    movel([0.122327, -1.228329, -2.662622, -0.821438, 1.570796, 1.693123],accel_mss,speed_ms,0,blend_radius_m)
    movel([0.122064, -1.229821, -2.661862, -0.820705, 1.570796, 1.692861],accel_mss,speed_ms,0,blend_radius_m)
    movel([0.121775, -1.231117, -2.661201, -0.820072, 1.570796, 1.692571],accel_mss,speed_ms,0,blend_radius_m)
    movel([0.121353, -1.232704, -2.660387, -0.819297, 1.570796, 1.692149],accel_mss,speed_ms,0,blend_radius_m)
    movel([0.120445, -1.235790, -2.658798, -0.817801, 1.570796, 1.691242],accel_mss,speed_ms,0,blend_radius_m)
    speed_ms = 0.003
    movel([0.120445, -1.239413, -2.660528, -0.812448, 1.570796, 1.691242],accel_mss,speed_ms,0,blend_radius_m)
    speed_ms = 0.007
    movel([0.119507, -1.242259, -2.659045, -0.811085, 1.570796, 1.690304],accel_mss,speed_ms,0,blend_radius_m)
    movel([0.118536, -1.244874, -2.657674, -0.809842, 1.570796, 1.689333],accel_mss,speed_ms,0,blend_radius_m)
    movel([0.117534, -1.247261, -2.656415, -0.808713, 1.570796, 1.688331],accel_mss,speed_ms,0,blend_radius_m)
    movel([0.117009, -1.248417, -2.655802, -0.808169, 1.570796, 1.687805],accel_mss,speed_ms,0,blend_radius_m)
    movel([0.116695, -1.249022, -2.655481, -0.807885, 1.570796, 1.687491],accel_mss,speed_ms,0,blend_radius_m)
    movel([0.116436, -1.249403, -2.655279, -0.807707, 1.570796, 1.687232],accel_mss,speed_ms,0,blend_radius_m)
    movel([0.116154, -1.249681, -2.655131, -0.807576, 1.570796, 1.686950],accel_mss,speed_ms,0,blend_radius_m)
    movel([0.114416, -1.250711, -2.654583, -0.807095, 1.570796, 1.685212],accel_mss,speed_ms,0,blend_radius_m)
    movel([0.110469, -1.252305, -2.653732, -0.806351, 1.570796, 1.681265],accel_mss,speed_ms,0,blend_radius_m)
    movel([0.105892, -1.253965, -2.652843, -0.805581, 1.570796, 1.676688],accel_mss,speed_ms,0,blend_radius_m)
    movel([0.101275, -1.255432, -2.652054, -0.804903, 1.570796, 1.672071],accel_mss,speed_ms,0,blend_radius_m)
    movel([0.097010, -1.256607, -2.651420, -0.804361, 1.570796, 1.667806],accel_mss,speed_ms,0,blend_radius_m)
    movel([0.093314, -1.257431, -2.650975, -0.803983, 1.570796, 1.664111],accel_mss,speed_ms,0,blend_radius_m)
    movel([0.090388, -1.257913, -2.650714, -0.803762, 1.570796, 1.661185],accel_mss,speed_ms,0,blend_radius_m)
    movel([0.089540, -1.257658, -2.650852, -0.803879, 1.570796, 1.660336],accel_mss,speed_ms,0,blend_radius_m)
    movel([0.088883, -1.255617, -2.651955, -0.804818, 1.570796, 1.659679],accel_mss,speed_ms,0,blend_radius_m)
    movel([0.089050, -1.247881, -2.656087, -0.808421, 1.570796, 1.659846],accel_mss,speed_ms,0,blend_radius_m)
    movel([0.089536, -1.239986, -2.660230, -0.812173, 1.570796, 1.660332],accel_mss,speed_ms,0,blend_radius_m)
    movel([0.090414, -1.234541, -2.663045, -0.814803, 1.570796, 1.661211],accel_mss,speed_ms,0,blend_radius_m)
    movel([0.090708, -1.233537, -2.663560, -0.815292, 1.570796, 1.661505],accel_mss,speed_ms,0,blend_radius_m)
    movel([0.091054, -1.232965, -2.663853, -0.815571, 1.570796, 1.661850],accel_mss,speed_ms,0,blend_radius_m)
    movel([0.091650, -1.232455, -2.664114, -0.815820, 1.570796, 1.662446],accel_mss,speed_ms,0,blend_radius_m)
    movel([0.093003, -1.231626, -2.664538, -0.816226, 1.570796, 1.663799],accel_mss,speed_ms,0,blend_radius_m)
    movel([0.095187, -1.230416, -2.665154, -0.816819, 1.570796, 1.665983],accel_mss,speed_ms,0,blend_radius_m)
    movel([0.097230, -1.229430, -2.665656, -0.817304, 1.570796, 1.668026],accel_mss,speed_ms,0,blend_radius_m)
    movel([0.099701, -1.228404, -2.666176, -0.817809, 1.570796, 1.670497],accel_mss,speed_ms,0,blend_radius_m)
    movel([0.103416, -1.227010, -2.666881, -0.818498, 1.570796, 1.674212],accel_mss,speed_ms,0,blend_radius_m)
    movel([0.108750, -1.225175, -2.667806, -0.819408, 1.570796, 1.679546],accel_mss,speed_ms,0,blend_radius_m)
    movel([0.113497, -1.223771, -2.668511, -0.820108, 1.570796, 1.684294],accel_mss,speed_ms,0,blend_radius_m)
    movel([0.117730, -1.222780, -2.669007, -0.820602, 1.570796, 1.688526],accel_mss,speed_ms,0,blend_radius_m)
    movel([0.121518, -1.222181, -2.669306, -0.820902, 1.570796, 1.692314],accel_mss,speed_ms,0,blend_radius_m)
    movel([0.122546, -1.222114, -2.669340, -0.820935, 1.570796, 1.693342],accel_mss,speed_ms,0,blend_radius_m)
    movel([0.122998, -1.222262, -2.669266, -0.820861, 1.570796, 1.693794],accel_mss,speed_ms,0,blend_radius_m)
    movel([0.123197, -1.222684, -2.669055, -0.820650, 1.570796, 1.693993],accel_mss,speed_ms,0,blend_radius_m)
    movel([0.123242, -1.223715, -2.668539, -0.820135, 1.570796, 1.694038],accel_mss,speed_ms,0,blend_radius_m)
    movel([0.123245, -1.224244, -2.668274, -0.819872, 1.570796, 1.694042],accel_mss,speed_ms,0,blend_radius_m)
    movel([0.123250, -1.224722, -2.668033, -0.819633, 1.570796, 1.694046],accel_mss,speed_ms,0,blend_radius_m)
    movel([0.123256, -1.225120, -2.667833, -0.819435, 1.570796, 1.694052],accel_mss,speed_ms,0,blend_radius_m)
    movel([0.123267, -1.225404, -2.667691, -0.819294, 1.570796, 1.694063],accel_mss,speed_ms,0,blend_radius_m)
    movel([0.123104, -1.226608, -2.667084, -0.818697, 1.570796, 1.693901],accel_mss,speed_ms,0,blend_radius_m)
    movel([0.122915, -1.227989, -2.666386, -0.818014, 1.570796, 1.693712],accel_mss,speed_ms,0,blend_radius_m)
    movel([0.122686, -1.229588, -2.665575, -0.817226, 1.570796, 1.693482],accel_mss,speed_ms,0,blend_radius_m)
    movel([0.122327, -1.231965, -2.664364, -0.816060, 1.570796, 1.693123],accel_mss,speed_ms,0,blend_radius_m)
    movel([0.122064, -1.233455, -2.663602, -0.815332, 1.570796, 1.692861],accel_mss,speed_ms,0,blend_radius_m)
    movel([0.121775, -1.234748, -2.662939, -0.814703, 1.570796, 1.692571],accel_mss,speed_ms,0,blend_radius_m)
    movel([0.121353, -1.236333, -2.662123, -0.813934, 1.570796, 1.692149],accel_mss,speed_ms,0,blend_radius_m)
    movel([0.120445, -1.239413, -2.660528, -0.812448, 1.570796, 1.691242],accel_mss,speed_ms,0,blend_radius_m)
    speed_ms = 0.003
    movel([0.120445, -1.225115, -2.653559, -0.833714, 1.570796, 1.691242],accel_mss,speed_ms,0,blend_radius_m)
    speed_ms = 1.000
    movel([0.120445, -1.198045, -2.639248, -0.875095, 1.570796, 1.691242],accel_mss,speed_ms,0,blend_radius_m)
    movel([0.119134, -1.211134, -2.632724, -0.868530, 1.570796, 1.689930],accel_mss,speed_ms,0,blend_radius_m)
    movel([0.119134, -1.238074, -2.646863, -0.827452, 1.570796, 1.689930],accel_mss,speed_ms,0,blend_radius_m)
    speed_ms = 0.003
    movel([0.119134, -1.248685, -2.652035, -0.811669, 1.570796, 1.689930],accel_mss,speed_ms,0,blend_radius_m)
    speed_ms = 0.007
    movel([0.119613, -1.248514, -2.652126, -0.811749, 1.570796, 1.690410],accel_mss,speed_ms,0,blend_radius_m)
    movel([0.120288, -1.248305, -2.652237, -0.811847, 1.570796, 1.691084],accel_mss,speed_ms,0,blend_radius_m)
    movel([0.121252, -1.248036, -2.652380, -0.811973, 1.570796, 1.692048],accel_mss,speed_ms,0,blend_radius_m)
    movel([0.122082, -1.247811, -2.652500, -0.812078, 1.570796, 1.692879],accel_mss,speed_ms,0,blend_radius_m)
    movel([0.122838, -1.247602, -2.652610, -0.812176, 1.570796, 1.693634],accel_mss,speed_ms,0,blend_radius_m)
    movel([0.123475, -1.247426, -2.652704, -0.812259, 1.570796, 1.694272],accel_mss,speed_ms,0,blend_radius_m)
    movel([0.124143, -1.247295, -2.652773, -0.812320, 1.570796, 1.694939],accel_mss,speed_ms,0,blend_radius_m)
    movel([0.124365, -1.247460, -2.652686, -0.812243, 1.570796, 1.695162],accel_mss,speed_ms,0,blend_radius_m)
    movel([0.124402, -1.247921, -2.652442, -0.812027, 1.570796, 1.695199],accel_mss,speed_ms,0,blend_radius_m)
    movel([0.124242, -1.248885, -2.651929, -0.811575, 1.570796, 1.695039],accel_mss,speed_ms,0,blend_radius_m)
    movel([0.124101, -1.249513, -2.651594, -0.811282, 1.570796, 1.694897],accel_mss,speed_ms,0,blend_radius_m)
    movel([0.123892, -1.250271, -2.651190, -0.810928, 1.570796, 1.694688],accel_mss,speed_ms,0,blend_radius_m)
    movel([0.123656, -1.251037, -2.650780, -0.810572, 1.570796, 1.694453],accel_mss,speed_ms,0,blend_radius_m)
    movel([0.123426, -1.251690, -2.650431, -0.810268, 1.570796, 1.694222],accel_mss,speed_ms,0,blend_radius_m)
    movel([0.122892, -1.252969, -2.649744, -0.809675, 1.570796, 1.693688],accel_mss,speed_ms,0,blend_radius_m)
    movel([0.122475, -1.253530, -2.649443, -0.809416, 1.570796, 1.693271],accel_mss,speed_ms,0,blend_radius_m)
    movel([0.121856, -1.253929, -2.649229, -0.809232, 1.570796, 1.692652],accel_mss,speed_ms,0,blend_radius_m)
    movel([0.120346, -1.254514, -2.648913, -0.808962, 1.570796, 1.691142],accel_mss,speed_ms,0,blend_radius_m)
    movel([0.119442, -1.254834, -2.648741, -0.808814, 1.570796, 1.690239],accel_mss,speed_ms,0,blend_radius_m)
    movel([0.118839, -1.255024, -2.648638, -0.808727, 1.570796, 1.689635],accel_mss,speed_ms,0,blend_radius_m)
    movel([0.118432, -1.255127, -2.648583, -0.808679, 1.570796, 1.689228],accel_mss,speed_ms,0,blend_radius_m)
    movel([0.118168, -1.254986, -2.648659, -0.808744, 1.570796, 1.688964],accel_mss,speed_ms,0,blend_radius_m)
    movel([0.118162, -1.254671, -2.648828, -0.808889, 1.570796, 1.688958],accel_mss,speed_ms,0,blend_radius_m)
    movel([0.118223, -1.254120, -2.649125, -0.809143, 1.570796, 1.689019],accel_mss,speed_ms,0,blend_radius_m)
    movel([0.118394, -1.253069, -2.649691, -0.809629, 1.570796, 1.689190],accel_mss,speed_ms,0,blend_radius_m)
    movel([0.118522, -1.252242, -2.650135, -0.810012, 1.570796, 1.689318],accel_mss,speed_ms,0,blend_radius_m)
    movel([0.118632, -1.251377, -2.650599, -0.810414, 1.570796, 1.689429],accel_mss,speed_ms,0,blend_radius_m)
    movel([0.118710, -1.250595, -2.651017, -0.810777, 1.570796, 1.689506],accel_mss,speed_ms,0,blend_radius_m)
    movel([0.118739, -1.250054, -2.651306, -0.811030, 1.570796, 1.689536],accel_mss,speed_ms,0,blend_radius_m)
    movel([0.118758, -1.249526, -2.651587, -0.811276, 1.570796, 1.689555],accel_mss,speed_ms,0,blend_radius_m)
    movel([0.118795, -1.249184, -2.651769, -0.811435, 1.570796, 1.689591],accel_mss,speed_ms,0,blend_radius_m)
    movel([0.118957, -1.248800, -2.651974, -0.811615, 1.570796, 1.689753],accel_mss,speed_ms,0,blend_radius_m)
    speed_ms = 0.003
    movel([0.119134, -1.252285, -2.653743, -0.806361, 1.570796, 1.689930],accel_mss,speed_ms,0,blend_radius_m)
    speed_ms = 0.007
    movel([0.119613, -1.252114, -2.653835, -0.806441, 1.570796, 1.690410],accel_mss,speed_ms,0,blend_radius_m)
    movel([0.120288, -1.251906, -2.653946, -0.806538, 1.570796, 1.691084],accel_mss,speed_ms,0,blend_radius_m)
    movel([0.121252, -1.251637, -2.654090, -0.806663, 1.570796, 1.692048],accel_mss,speed_ms,0,blend_radius_m)
    movel([0.122082, -1.251413, -2.654209, -0.806767, 1.570796, 1.692879],accel_mss,speed_ms,0,blend_radius_m)
    movel([0.122838, -1.251204, -2.654320, -0.806864, 1.570796, 1.693634],accel_mss,speed_ms,0,blend_radius_m)
    movel([0.123475, -1.251028, -2.654414, -0.806947, 1.570796, 1.694272],accel_mss,speed_ms,0,blend_radius_m)
    movel([0.124143, -1.250898, -2.654484, -0.807008, 1.570796, 1.694939],accel_mss,speed_ms,0,blend_radius_m)
    movel([0.124365, -1.251062, -2.654396, -0.806931, 1.570796, 1.695162],accel_mss,speed_ms,0,blend_radius_m)
    movel([0.124402, -1.251522, -2.654151, -0.806716, 1.570796, 1.695199],accel_mss,speed_ms,0,blend_radius_m)
    movel([0.124242, -1.252485, -2.653636, -0.806268, 1.570796, 1.695039],accel_mss,speed_ms,0,blend_radius_m)
    movel([0.124101, -1.253111, -2.653301, -0.805977, 1.570796, 1.694897],accel_mss,speed_ms,0,blend_radius_m)
    movel([0.123892, -1.253868, -2.652895, -0.805626, 1.570796, 1.694688],accel_mss,speed_ms,0,blend_radius_m)
    movel([0.123656, -1.254633, -2.652484, -0.805272, 1.570796, 1.694453],accel_mss,speed_ms,0,blend_radius_m)
    movel([0.123426, -1.255284, -2.652134, -0.804971, 1.570796, 1.694222],accel_mss,speed_ms,0,blend_radius_m)
    movel([0.122892, -1.256561, -2.651445, -0.804383, 1.570796, 1.693688],accel_mss,speed_ms,0,blend_radius_m)
    movel([0.122475, -1.257121, -2.651143, -0.804125, 1.570796, 1.693271],accel_mss,speed_ms,0,blend_radius_m)
    movel([0.121856, -1.257519, -2.650927, -0.803943, 1.570796, 1.692652],accel_mss,speed_ms,0,blend_radius_m)
    movel([0.120346, -1.258103, -2.650611, -0.803675, 1.570796, 1.691142],accel_mss,speed_ms,0,blend_radius_m)
    movel([0.119442, -1.258422, -2.650438, -0.803529, 1.570796, 1.690239],accel_mss,speed_ms,0,blend_radius_m)
    movel([0.118839, -1.258612, -2.650335, -0.803442, 1.570796, 1.689635],accel_mss,speed_ms,0,blend_radius_m)
    movel([0.118432, -1.258715, -2.650279, -0.803395, 1.570796, 1.689228],accel_mss,speed_ms,0,blend_radius_m)
    movel([0.118168, -1.258574, -2.650356, -0.803459, 1.570796, 1.688964],accel_mss,speed_ms,0,blend_radius_m)
    movel([0.118162, -1.258260, -2.650526, -0.803603, 1.570796, 1.688958],accel_mss,speed_ms,0,blend_radius_m)
    movel([0.118223, -1.257710, -2.650824, -0.803855, 1.570796, 1.689019],accel_mss,speed_ms,0,blend_radius_m)
    movel([0.118394, -1.256660, -2.651392, -0.804337, 1.570796, 1.689190],accel_mss,speed_ms,0,blend_radius_m)
    movel([0.118522, -1.255835, -2.651837, -0.804717, 1.570796, 1.689318],accel_mss,speed_ms,0,blend_radius_m)
    movel([0.118632, -1.254971, -2.652302, -0.805116, 1.570796, 1.689429],accel_mss,speed_ms,0,blend_radius_m)
    movel([0.118710, -1.254191, -2.652721, -0.805476, 1.570796, 1.689506],accel_mss,speed_ms,0,blend_radius_m)
    movel([0.118739, -1.253651, -2.653011, -0.805727, 1.570796, 1.689536],accel_mss,speed_ms,0,blend_radius_m)
    movel([0.118758, -1.253124, -2.653294, -0.805971, 1.570796, 1.689555],accel_mss,speed_ms,0,blend_radius_m)
    movel([0.118795, -1.252783, -2.653477, -0.806130, 1.570796, 1.689591],accel_mss,speed_ms,0,blend_radius_m)
    movel([0.118957, -1.252400, -2.653682, -0.806308, 1.570796, 1.689753],accel_mss,speed_ms,0,blend_radius_m)
    speed_ms = 0.003
    movel([0.119134, -1.238074, -2.646863, -0.827452, 1.570796, 1.689930],accel_mss,speed_ms,0,blend_radius_m)
    speed_ms = 1.000
    movel([0.119134, -1.211134, -2.632724, -0.868530, 1.570796, 1.689930],accel_mss,speed_ms,0,blend_radius_m)
    movel([0.110419, -1.221617, -2.627362, -0.863409, 1.570796, 1.681215],accel_mss,speed_ms,0,blend_radius_m)
    movel([0.110419, -1.248444, -2.641362, -0.822583, 1.570796, 1.681215],accel_mss,speed_ms,0,blend_radius_m)
    speed_ms = 0.003
    movel([0.110419, -1.259001, -2.646482, -0.806906, 1.570796, 1.681215],accel_mss,speed_ms,0,blend_radius_m)
    speed_ms = 0.007
    movel([0.110103, -1.259367, -2.646283, -0.806739, 1.570796, 1.680899],accel_mss,speed_ms,0,blend_radius_m)
    movel([0.109738, -1.259520, -2.646199, -0.806670, 1.570796, 1.680535],accel_mss,speed_ms,0,blend_radius_m)
    movel([0.109218, -1.259703, -2.646100, -0.806586, 1.570796, 1.680015],accel_mss,speed_ms,0,blend_radius_m)
    movel([0.108623, -1.259897, -2.645994, -0.806498, 1.570796, 1.679419],accel_mss,speed_ms,0,blend_radius_m)
    movel([0.108306, -1.259974, -2.645952, -0.806463, 1.570796, 1.679103],accel_mss,speed_ms,0,blend_radius_m)
    movel([0.108167, -1.259780, -2.646058, -0.806552, 1.570796, 1.678963],accel_mss,speed_ms,0,blend_radius_m)
    movel([0.108618, -1.259522, -2.646198, -0.806669, 1.570796, 1.679415],accel_mss,speed_ms,0,blend_radius_m)
    movel([0.109124, -1.259324, -2.646306, -0.806759, 1.570796, 1.679920],accel_mss,speed_ms,0,blend_radius_m)
    movel([0.109843, -1.259068, -2.646446, -0.806875, 1.570796, 1.680640],accel_mss,speed_ms,0,blend_radius_m)
    movel([0.110242, -1.258971, -2.646499, -0.806920, 1.570796, 1.681039],accel_mss,speed_ms,0,blend_radius_m)
    speed_ms = 0.003
    movel([0.110419, -1.262581, -2.648172, -0.801635, 1.570796, 1.681215],accel_mss,speed_ms,0,blend_radius_m)
    speed_ms = 0.007
    movel([0.110103, -1.262947, -2.647972, -0.801470, 1.570796, 1.680899],accel_mss,speed_ms,0,blend_radius_m)
    movel([0.109738, -1.263099, -2.647889, -0.801401, 1.570796, 1.680535],accel_mss,speed_ms,0,blend_radius_m)
    movel([0.109218, -1.263282, -2.647789, -0.801318, 1.570796, 1.680015],accel_mss,speed_ms,0,blend_radius_m)
    movel([0.108623, -1.263476, -2.647683, -0.801231, 1.570796, 1.679419],accel_mss,speed_ms,0,blend_radius_m)
    movel([0.108306, -1.263553, -2.647640, -0.801196, 1.570796, 1.679103],accel_mss,speed_ms,0,blend_radius_m)
    movel([0.108167, -1.263358, -2.647747, -0.801284, 1.570796, 1.678963],accel_mss,speed_ms,0,blend_radius_m)
    movel([0.108618, -1.263101, -2.647888, -0.801400, 1.570796, 1.679415],accel_mss,speed_ms,0,blend_radius_m)
    movel([0.109124, -1.262903, -2.647996, -0.801490, 1.570796, 1.679920],accel_mss,speed_ms,0,blend_radius_m)
    movel([0.109843, -1.262648, -2.648136, -0.801605, 1.570796, 1.680640],accel_mss,speed_ms,0,blend_radius_m)
    movel([0.110242, -1.262551, -2.648189, -0.801649, 1.570796, 1.681039],accel_mss,speed_ms,0,blend_radius_m)
    speed_ms = 0.003
    movel([0.110419, -1.248444, -2.641362, -0.822583, 1.570796, 1.681215],accel_mss,speed_ms,0,blend_radius_m)
    speed_ms = 1.000
    movel([0.110419, -1.221617, -2.627362, -0.863409, 1.570796, 1.681215],accel_mss,speed_ms,0,blend_radius_m)
    movel([0.110927, -1.220864, -2.627752, -0.863773, 1.570796, 1.681724],accel_mss,speed_ms,0,blend_radius_m)
    movel([0.110927, -1.247699, -2.641762, -0.822928, 1.570796, 1.681724],accel_mss,speed_ms,0,blend_radius_m)
    speed_ms = 0.003
    movel([0.110927, -1.258260, -2.646885, -0.807244, 1.570796, 1.681724],accel_mss,speed_ms,0,blend_radius_m)
    speed_ms = 0.007
    movel([0.111162, -1.258336, -2.646844, -0.807209, 1.570796, 1.681958],accel_mss,speed_ms,0,blend_radius_m)
    movel([0.111335, -1.258610, -2.646695, -0.807084, 1.570796, 1.682131],accel_mss,speed_ms,0,blend_radius_m)
    movel([0.111245, -1.259072, -2.646443, -0.806873, 1.570796, 1.682041],accel_mss,speed_ms,0,blend_radius_m)
    movel([0.110931, -1.259552, -2.646182, -0.806655, 1.570796, 1.681728],accel_mss,speed_ms,0,blend_radius_m)
    movel([0.110499, -1.259877, -2.646005, -0.806507, 1.570796, 1.681295],accel_mss,speed_ms,0,blend_radius_m)
    movel([0.110195, -1.260124, -2.645870, -0.806395, 1.570796, 1.680991],accel_mss,speed_ms,0,blend_radius_m)
    movel([0.109991, -1.260507, -2.645661, -0.806221, 1.570796, 1.680787],accel_mss,speed_ms,0,blend_radius_m)
    movel([0.109819, -1.261212, -2.645275, -0.805902, 1.570796, 1.680615],accel_mss,speed_ms,0,blend_radius_m)
    movel([0.109528, -1.262982, -2.644305, -0.805102, 1.570796, 1.680325],accel_mss,speed_ms,0,blend_radius_m)
    movel([0.109349, -1.264046, -2.643719, -0.804623, 1.570796, 1.680145],accel_mss,speed_ms,0,blend_radius_m)
    movel([0.109167, -1.264994, -2.643197, -0.804198, 1.570796, 1.679964],accel_mss,speed_ms,0,blend_radius_m)
    movel([0.108999, -1.265794, -2.642755, -0.803840, 1.570796, 1.679795],accel_mss,speed_ms,0,blend_radius_m)
    movel([0.108635, -1.266395, -2.642422, -0.803571, 1.570796, 1.679431],accel_mss,speed_ms,0,blend_radius_m)
    movel([0.108350, -1.266617, -2.642300, -0.803472, 1.570796, 1.679146],accel_mss,speed_ms,0,blend_radius_m)
    movel([0.108060, -1.266674, -2.642268, -0.803447, 1.570796, 1.678857],accel_mss,speed_ms,0,blend_radius_m)
    movel([0.107768, -1.266569, -2.642326, -0.803494, 1.570796, 1.678564],accel_mss,speed_ms,0,blend_radius_m)
    movel([0.107626, -1.266380, -2.642431, -0.803578, 1.570796, 1.678423],accel_mss,speed_ms,0,blend_radius_m)
    movel([0.107594, -1.266055, -2.642611, -0.803723, 1.570796, 1.678390],accel_mss,speed_ms,0,blend_radius_m)
    movel([0.107658, -1.265425, -2.642959, -0.804005, 1.570796, 1.678455],accel_mss,speed_ms,0,blend_radius_m)
    movel([0.107927, -1.263671, -2.643926, -0.804792, 1.570796, 1.678724],accel_mss,speed_ms,0,blend_radius_m)
    movel([0.108213, -1.261753, -2.644979, -0.805657, 1.570796, 1.679010],accel_mss,speed_ms,0,blend_radius_m)
    movel([0.108244, -1.261039, -2.645370, -0.805980, 1.570796, 1.679041],accel_mss,speed_ms,0,blend_radius_m)
    movel([0.108086, -1.260774, -2.645515, -0.806100, 1.570796, 1.678882],accel_mss,speed_ms,0,blend_radius_m)
    movel([0.107730, -1.260767, -2.645519, -0.806103, 1.570796, 1.678526],accel_mss,speed_ms,0,blend_radius_m)
    movel([0.107264, -1.260711, -2.645549, -0.806129, 1.570796, 1.678061],accel_mss,speed_ms,0,blend_radius_m)
    movel([0.107166, -1.260236, -2.645809, -0.806344, 1.570796, 1.677963],accel_mss,speed_ms,0,blend_radius_m)
    movel([0.107499, -1.259585, -2.646164, -0.806640, 1.570796, 1.678295],accel_mss,speed_ms,0,blend_radius_m)
    movel([0.108088, -1.259128, -2.646413, -0.806848, 1.570796, 1.678884],accel_mss,speed_ms,0,blend_radius_m)
    movel([0.108427, -1.258906, -2.646534, -0.806949, 1.570796, 1.679223],accel_mss,speed_ms,0,blend_radius_m)
    movel([0.108679, -1.258608, -2.646696, -0.807085, 1.570796, 1.679475],accel_mss,speed_ms,0,blend_radius_m)
    movel([0.108908, -1.258251, -2.646890, -0.807248, 1.570796, 1.679704],accel_mss,speed_ms,0,blend_radius_m)
    movel([0.109183, -1.257900, -2.647081, -0.807408, 1.570796, 1.679979],accel_mss,speed_ms,0,blend_radius_m)
    movel([0.109450, -1.257617, -2.647235, -0.807537, 1.570796, 1.680246],accel_mss,speed_ms,0,blend_radius_m)
    movel([0.109811, -1.257500, -2.647298, -0.807591, 1.570796, 1.680607],accel_mss,speed_ms,0,blend_radius_m)
    movel([0.110051, -1.257638, -2.647223, -0.807528, 1.570796, 1.680848],accel_mss,speed_ms,0,blend_radius_m)
    movel([0.110266, -1.257831, -2.647118, -0.807440, 1.570796, 1.681062],accel_mss,speed_ms,0,blend_radius_m)
    movel([0.110377, -1.258036, -2.647007, -0.807346, 1.570796, 1.681173],accel_mss,speed_ms,0,blend_radius_m)
    movel([0.110587, -1.258217, -2.646908, -0.807263, 1.570796, 1.681383],accel_mss,speed_ms,0,blend_radius_m)
    movel([0.110927, -1.258260, -2.646885, -0.807244, 1.570796, 1.681724],accel_mss,speed_ms,0,blend_radius_m)
    speed_ms = 0.003
    movel([0.110927, -1.261842, -2.648577, -0.801970, 1.570796, 1.681724],accel_mss,speed_ms,0,blend_radius_m)
    speed_ms = 0.007
    movel([0.111162, -1.261917, -2.648535, -0.801936, 1.570796, 1.681958],accel_mss,speed_ms,0,blend_radius_m)
    movel([0.111335, -1.262191, -2.648386, -0.801812, 1.570796, 1.682131],accel_mss,speed_ms,0,blend_radius_m)
    movel([0.111245, -1.262652, -2.648134, -0.801603, 1.570796, 1.682041],accel_mss,speed_ms,0,blend_radius_m)
    movel([0.110931, -1.263131, -2.647871, -0.801387, 1.570796, 1.681728],accel_mss,speed_ms,0,blend_radius_m)
    movel([0.110499, -1.263456, -2.647693, -0.801240, 1.570796, 1.681295],accel_mss,speed_ms,0,blend_radius_m)
    movel([0.110195, -1.263702, -2.647558, -0.801129, 1.570796, 1.680991],accel_mss,speed_ms,0,blend_radius_m)
    movel([0.109991, -1.264084, -2.647349, -0.800956, 1.570796, 1.680787],accel_mss,speed_ms,0,blend_radius_m)
    movel([0.109819, -1.264788, -2.646962, -0.800639, 1.570796, 1.680615],accel_mss,speed_ms,0,blend_radius_m)
    movel([0.109528, -1.266554, -2.645988, -0.799846, 1.570796, 1.680325],accel_mss,speed_ms,0,blend_radius_m)
    movel([0.109349, -1.267617, -2.645401, -0.799371, 1.570796, 1.680145],accel_mss,speed_ms,0,blend_radius_m)
    movel([0.109167, -1.268562, -2.644877, -0.798950, 1.570796, 1.679964],accel_mss,speed_ms,0,blend_radius_m)
    movel([0.108999, -1.269361, -2.644434, -0.798594, 1.570796, 1.679795],accel_mss,speed_ms,0,blend_radius_m)
    movel([0.108635, -1.269961, -2.644100, -0.798328, 1.570796, 1.679431],accel_mss,speed_ms,0,blend_radius_m)
    movel([0.108350, -1.270182, -2.643977, -0.798230, 1.570796, 1.679146],accel_mss,speed_ms,0,blend_radius_m)
    movel([0.108060, -1.270239, -2.643945, -0.798204, 1.570796, 1.678857],accel_mss,speed_ms,0,blend_radius_m)
    movel([0.107768, -1.270135, -2.644003, -0.798251, 1.570796, 1.678564],accel_mss,speed_ms,0,blend_radius_m)
    movel([0.107626, -1.269946, -2.644109, -0.798335, 1.570796, 1.678423],accel_mss,speed_ms,0,blend_radius_m)
    movel([0.107594, -1.269621, -2.644289, -0.798479, 1.570796, 1.678390],accel_mss,speed_ms,0,blend_radius_m)
    movel([0.107658, -1.268993, -2.644638, -0.798758, 1.570796, 1.678455],accel_mss,speed_ms,0,blend_radius_m)
    movel([0.107927, -1.267242, -2.645608, -0.799538, 1.570796, 1.678724],accel_mss,speed_ms,0,blend_radius_m)
    movel([0.108213, -1.265328, -2.646665, -0.800397, 1.570796, 1.679010],accel_mss,speed_ms,0,blend_radius_m)
    movel([0.108244, -1.264615, -2.647057, -0.800717, 1.570796, 1.679041],accel_mss,speed_ms,0,blend_radius_m)
    movel([0.108086, -1.264350, -2.647202, -0.800836, 1.570796, 1.678882],accel_mss,speed_ms,0,blend_radius_m)
    movel([0.107730, -1.264344, -2.647206, -0.800839, 1.570796, 1.678526],accel_mss,speed_ms,0,blend_radius_m)
    movel([0.107264, -1.264288, -2.647237, -0.800865, 1.570796, 1.678061],accel_mss,speed_ms,0,blend_radius_m)
    movel([0.107166, -1.263814, -2.647497, -0.801078, 1.570796, 1.677963],accel_mss,speed_ms,0,blend_radius_m)
    movel([0.107499, -1.263164, -2.647853, -0.801372, 1.570796, 1.678295],accel_mss,speed_ms,0,blend_radius_m)
    movel([0.108088, -1.262708, -2.648103, -0.801578, 1.570796, 1.678884],accel_mss,speed_ms,0,blend_radius_m)
    movel([0.108427, -1.262486, -2.648224, -0.801678, 1.570796, 1.679223],accel_mss,speed_ms,0,blend_radius_m)
    movel([0.108679, -1.262189, -2.648387, -0.801813, 1.570796, 1.679475],accel_mss,speed_ms,0,blend_radius_m)
    movel([0.108908, -1.261832, -2.648582, -0.801975, 1.570796, 1.679704],accel_mss,speed_ms,0,blend_radius_m)
    movel([0.109183, -1.261482, -2.648773, -0.802133, 1.570796, 1.679979],accel_mss,speed_ms,0,blend_radius_m)
    movel([0.109450, -1.261200, -2.648927, -0.802262, 1.570796, 1.680246],accel_mss,speed_ms,0,blend_radius_m)
    movel([0.109811, -1.261083, -2.648991, -0.802315, 1.570796, 1.680607],accel_mss,speed_ms,0,blend_radius_m)
    movel([0.110051, -1.261221, -2.648916, -0.802252, 1.570796, 1.680848],accel_mss,speed_ms,0,blend_radius_m)
    movel([0.110266, -1.261413, -2.648811, -0.802165, 1.570796, 1.681062],accel_mss,speed_ms,0,blend_radius_m)
    movel([0.110377, -1.261618, -2.648699, -0.802072, 1.570796, 1.681173],accel_mss,speed_ms,0,blend_radius_m)
    movel([0.110587, -1.261799, -2.648600, -0.801990, 1.570796, 1.681383],accel_mss,speed_ms,0,blend_radius_m)
    movel([0.110927, -1.261842, -2.648577, -0.801970, 1.570796, 1.681724],accel_mss,speed_ms,0,blend_radius_m)
    speed_ms = 0.003
    movel([0.110927, -1.247699, -2.641762, -0.822928, 1.570796, 1.681724],accel_mss,speed_ms,0,blend_radius_m)
    speed_ms = 1.000
    movel([0.110927, -1.220864, -2.627752, -0.863773, 1.570796, 1.681724],accel_mss,speed_ms,0,blend_radius_m)
    movel([0.111880, -1.220520, -2.627929, -0.863940, 1.570796, 1.682676],accel_mss,speed_ms,0,blend_radius_m)
    movel([0.111880, -1.247359, -2.641944, -0.823086, 1.570796, 1.682676],accel_mss,speed_ms,0,blend_radius_m)
    speed_ms = 0.003
    movel([0.111880, -1.257921, -2.647069, -0.807398, 1.570796, 1.682676],accel_mss,speed_ms,0,blend_radius_m)
    speed_ms = 0.007
    movel([0.111646, -1.259471, -2.646226, -0.806692, 1.570796, 1.682442],accel_mss,speed_ms,0,blend_radius_m)
    movel([0.111379, -1.261243, -2.645258, -0.805888, 1.570796, 1.682175],accel_mss,speed_ms,0,blend_radius_m)
    movel([0.111116, -1.263008, -2.644290, -0.805090, 1.570796, 1.681913],accel_mss,speed_ms,0,blend_radius_m)
    movel([0.110781, -1.265207, -2.643080, -0.804103, 1.570796, 1.681578],accel_mss,speed_ms,0,blend_radius_m)
    movel([0.110564, -1.266458, -2.642388, -0.803543, 1.570796, 1.681360],accel_mss,speed_ms,0,blend_radius_m)
    movel([0.110395, -1.267274, -2.641935, -0.803179, 1.570796, 1.681191],accel_mss,speed_ms,0,blend_radius_m)
    movel([0.110254, -1.267551, -2.641782, -0.803056, 1.570796, 1.681050],accel_mss,speed_ms,0,blend_radius_m)
    movel([0.109445, -1.267985, -2.641541, -0.802863, 1.570796, 1.680241],accel_mss,speed_ms,0,blend_radius_m)
    movel([0.108456, -1.268322, -2.641354, -0.802714, 1.570796, 1.679252],accel_mss,speed_ms,0,blend_radius_m)
    movel([0.106110, -1.269067, -2.640939, -0.802383, 1.570796, 1.676906],accel_mss,speed_ms,0,blend_radius_m)
    movel([0.099234, -1.271239, -2.639727, -0.801423, 1.570796, 1.670030],accel_mss,speed_ms,0,blend_radius_m)
    movel([0.094434, -1.272745, -2.638883, -0.800761, 1.570796, 1.665230],accel_mss,speed_ms,0,blend_radius_m)
    movel([0.090679, -1.273913, -2.638226, -0.800250, 1.570796, 1.661475],accel_mss,speed_ms,0,blend_radius_m)
    movel([0.090382, -1.273921, -2.638222, -0.800247, 1.570796, 1.661178],accel_mss,speed_ms,0,blend_radius_m)
    movel([0.090308, -1.273275, -2.638585, -0.800529, 1.570796, 1.661104],accel_mss,speed_ms,0,blend_radius_m)
    movel([0.090387, -1.272418, -2.639066, -0.800905, 1.570796, 1.661183],accel_mss,speed_ms,0,blend_radius_m)
    movel([0.090598, -1.270730, -2.640011, -0.801648, 1.570796, 1.661394],accel_mss,speed_ms,0,blend_radius_m)
    movel([0.090772, -1.269448, -2.640727, -0.802214, 1.570796, 1.661569],accel_mss,speed_ms,0,blend_radius_m)
    movel([0.090933, -1.268415, -2.641302, -0.802672, 1.570796, 1.661730],accel_mss,speed_ms,0,blend_radius_m)
    movel([0.091081, -1.267562, -2.641776, -0.803051, 1.570796, 1.661878],accel_mss,speed_ms,0,blend_radius_m)
    movel([0.091342, -1.267303, -2.641919, -0.803166, 1.570796, 1.662139],accel_mss,speed_ms,0,blend_radius_m)
    movel([0.091673, -1.267392, -2.641870, -0.803127, 1.570796, 1.662469],accel_mss,speed_ms,0,blend_radius_m)
    movel([0.091927, -1.267417, -2.641856, -0.803116, 1.570796, 1.662723],accel_mss,speed_ms,0,blend_radius_m)
    movel([0.092311, -1.267404, -2.641864, -0.803122, 1.570796, 1.663108],accel_mss,speed_ms,0,blend_radius_m)
    movel([0.092453, -1.267633, -2.641737, -0.803020, 1.570796, 1.663250],accel_mss,speed_ms,0,blend_radius_m)
    movel([0.092461, -1.268193, -2.641425, -0.802771, 1.570796, 1.663257],accel_mss,speed_ms,0,blend_radius_m)
    movel([0.092320, -1.269424, -2.640740, -0.802225, 1.570796, 1.663116],accel_mss,speed_ms,0,blend_radius_m)
    movel([0.092175, -1.270710, -2.640023, -0.801656, 1.570796, 1.662971],accel_mss,speed_ms,0,blend_radius_m)
    movel([0.092201, -1.271259, -2.639715, -0.801414, 1.570796, 1.662997],accel_mss,speed_ms,0,blend_radius_m)
    movel([0.092385, -1.271465, -2.639600, -0.801324, 1.570796, 1.663181],accel_mss,speed_ms,0,blend_radius_m)
    movel([0.092744, -1.271444, -2.639612, -0.801333, 1.570796, 1.663541],accel_mss,speed_ms,0,blend_radius_m)
    movel([0.093158, -1.271191, -2.639754, -0.801445, 1.570796, 1.663954],accel_mss,speed_ms,0,blend_radius_m)
    movel([0.093440, -1.270802, -2.639971, -0.801616, 1.570796, 1.664237],accel_mss,speed_ms,0,blend_radius_m)
    movel([0.093651, -1.270128, -2.640347, -0.801913, 1.570796, 1.664448],accel_mss,speed_ms,0,blend_radius_m)
    movel([0.093890, -1.268782, -2.641098, -0.802509, 1.570796, 1.664686],accel_mss,speed_ms,0,blend_radius_m)
    movel([0.094066, -1.267708, -2.641695, -0.802986, 1.570796, 1.664863],accel_mss,speed_ms,0,blend_radius_m)
    movel([0.094187, -1.267166, -2.641995, -0.803227, 1.570796, 1.664983],accel_mss,speed_ms,0,blend_radius_m)
    movel([0.094304, -1.266842, -2.642175, -0.803372, 1.570796, 1.665100],accel_mss,speed_ms,0,blend_radius_m)
    movel([0.094576, -1.266568, -2.642327, -0.803494, 1.570796, 1.665372],accel_mss,speed_ms,0,blend_radius_m)
    movel([0.094860, -1.266356, -2.642444, -0.803589, 1.570796, 1.665657],accel_mss,speed_ms,0,blend_radius_m)
    movel([0.095215, -1.265979, -2.642653, -0.803757, 1.570796, 1.666012],accel_mss,speed_ms,0,blend_radius_m)
    movel([0.095415, -1.265557, -2.642886, -0.803946, 1.570796, 1.666211],accel_mss,speed_ms,0,blend_radius_m)
    movel([0.095501, -1.265189, -2.643089, -0.804111, 1.570796, 1.666298],accel_mss,speed_ms,0,blend_radius_m)
    movel([0.095460, -1.264959, -2.643216, -0.804214, 1.570796, 1.666256],accel_mss,speed_ms,0,blend_radius_m)
    movel([0.095278, -1.264822, -2.643292, -0.804275, 1.570796, 1.666075],accel_mss,speed_ms,0,blend_radius_m)
    movel([0.094918, -1.264756, -2.643328, -0.804305, 1.570796, 1.665714],accel_mss,speed_ms,0,blend_radius_m)
    movel([0.094621, -1.264580, -2.643425, -0.804384, 1.570796, 1.665417],accel_mss,speed_ms,0,blend_radius_m)
    movel([0.094596, -1.264324, -2.643566, -0.804498, 1.570796, 1.665392],accel_mss,speed_ms,0,blend_radius_m)
    movel([0.094629, -1.263697, -2.643912, -0.804780, 1.570796, 1.665426],accel_mss,speed_ms,0,blend_radius_m)
    movel([0.094635, -1.262961, -2.644316, -0.805111, 1.570796, 1.665432],accel_mss,speed_ms,0,blend_radius_m)
    movel([0.094510, -1.262579, -2.644526, -0.805284, 1.570796, 1.665306],accel_mss,speed_ms,0,blend_radius_m)
    movel([0.094243, -1.262479, -2.644581, -0.805329, 1.570796, 1.665039],accel_mss,speed_ms,0,blend_radius_m)
    movel([0.093835, -1.262614, -2.644507, -0.805268, 1.570796, 1.664631],accel_mss,speed_ms,0,blend_radius_m)
    movel([0.093555, -1.262823, -2.644392, -0.805174, 1.570796, 1.664352],accel_mss,speed_ms,0,blend_radius_m)
    movel([0.093224, -1.263474, -2.644034, -0.804881, 1.570796, 1.664020],accel_mss,speed_ms,0,blend_radius_m)
    movel([0.093066, -1.264195, -2.643638, -0.804557, 1.570796, 1.663862],accel_mss,speed_ms,0,blend_radius_m)
    movel([0.092919, -1.264835, -2.643285, -0.804270, 1.570796, 1.663715],accel_mss,speed_ms,0,blend_radius_m)
    movel([0.092764, -1.265200, -2.643083, -0.804106, 1.570796, 1.663561],accel_mss,speed_ms,0,blend_radius_m)
    movel([0.092248, -1.265595, -2.642865, -0.803929, 1.570796, 1.663044],accel_mss,speed_ms,0,blend_radius_m)
    movel([0.091948, -1.265768, -2.642769, -0.803851, 1.570796, 1.662744],accel_mss,speed_ms,0,blend_radius_m)
    movel([0.091695, -1.266027, -2.642626, -0.803736, 1.570796, 1.662491],accel_mss,speed_ms,0,blend_radius_m)
    movel([0.091391, -1.266296, -2.642477, -0.803616, 1.570796, 1.662187],accel_mss,speed_ms,0,blend_radius_m)
    movel([0.091166, -1.266089, -2.642592, -0.803708, 1.570796, 1.661962],accel_mss,speed_ms,0,blend_radius_m)
    movel([0.091445, -1.264045, -2.643720, -0.804624, 1.570796, 1.662241],accel_mss,speed_ms,0,blend_radius_m)
    movel([0.091760, -1.262004, -2.644841, -0.805543, 1.570796, 1.662556],accel_mss,speed_ms,0,blend_radius_m)
    movel([0.091988, -1.261594, -2.645066, -0.805729, 1.570796, 1.662785],accel_mss,speed_ms,0,blend_radius_m)
    movel([0.094110, -1.260792, -2.645505, -0.806092, 1.570796, 1.664907],accel_mss,speed_ms,0,blend_radius_m)
    movel([0.096668, -1.259933, -2.645974, -0.806482, 1.570796, 1.667464],accel_mss,speed_ms,0,blend_radius_m)
    movel([0.100580, -1.258657, -2.646670, -0.807063, 1.570796, 1.671376],accel_mss,speed_ms,0,blend_radius_m)
    movel([0.107027, -1.256592, -2.647790, -0.808007, 1.570796, 1.677824],accel_mss,speed_ms,0,blend_radius_m)
    movel([0.109986, -1.255677, -2.648286, -0.808427, 1.570796, 1.680783],accel_mss,speed_ms,0,blend_radius_m)
    movel([0.111807, -1.255142, -2.648574, -0.808672, 1.570796, 1.682603],accel_mss,speed_ms,0,blend_radius_m)
    movel([0.112142, -1.255147, -2.648572, -0.808670, 1.570796, 1.682938],accel_mss,speed_ms,0,blend_radius_m)
    movel([0.112198, -1.255613, -2.648320, -0.808456, 1.570796, 1.682994],accel_mss,speed_ms,0,blend_radius_m)
    movel([0.112144, -1.256155, -2.648027, -0.808207, 1.570796, 1.682940],accel_mss,speed_ms,0,blend_radius_m)
    movel([0.112026, -1.256971, -2.647585, -0.807833, 1.570796, 1.682822],accel_mss,speed_ms,0,blend_radius_m)
    movel([0.111880, -1.257921, -2.647069, -0.807398, 1.570796, 1.682676],accel_mss,speed_ms,0,blend_radius_m)
    speed_ms = 0.003
    movel([0.111880, -1.261504, -2.648761, -0.802124, 1.570796, 1.682676],accel_mss,speed_ms,0,blend_radius_m)
    speed_ms = 0.007
    movel([0.111646, -1.263051, -2.647915, -0.801423, 1.570796, 1.682442],accel_mss,speed_ms,0,blend_radius_m)
    movel([0.111379, -1.264819, -2.646945, -0.800625, 1.570796, 1.682175],accel_mss,speed_ms,0,blend_radius_m)
    movel([0.111116, -1.266581, -2.645974, -0.799835, 1.570796, 1.681913],accel_mss,speed_ms,0,blend_radius_m)
    movel([0.110781, -1.268775, -2.644759, -0.798855, 1.570796, 1.681578],accel_mss,speed_ms,0,blend_radius_m)
    movel([0.110564, -1.270024, -2.644065, -0.798300, 1.570796, 1.681360],accel_mss,speed_ms,0,blend_radius_m)
    movel([0.110395, -1.270838, -2.643611, -0.797939, 1.570796, 1.681191],accel_mss,speed_ms,0,blend_radius_m)
    movel([0.110254, -1.271114, -2.643458, -0.797817, 1.570796, 1.681050],accel_mss,speed_ms,0,blend_radius_m)
    movel([0.109445, -1.271547, -2.643216, -0.797626, 1.570796, 1.680241],accel_mss,speed_ms,0,blend_radius_m)
    movel([0.108456, -1.271883, -2.643028, -0.797477, 1.570796, 1.679252],accel_mss,speed_ms,0,blend_radius_m)
    movel([0.106110, -1.272627, -2.642613, -0.797150, 1.570796, 1.676906],accel_mss,speed_ms,0,blend_radius_m)
    movel([0.099234, -1.274795, -2.641396, -0.796198, 1.570796, 1.670030],accel_mss,speed_ms,0,blend_radius_m)
    movel([0.094434, -1.276298, -2.640549, -0.795542, 1.570796, 1.665230],accel_mss,speed_ms,0,blend_radius_m)
    movel([0.090679, -1.277464, -2.639891, -0.795035, 1.570796, 1.661475],accel_mss,speed_ms,0,blend_radius_m)
    movel([0.090382, -1.277471, -2.639887, -0.795031, 1.570796, 1.661178],accel_mss,speed_ms,0,blend_radius_m)
    movel([0.090308, -1.276827, -2.640251, -0.795311, 1.570796, 1.661104],accel_mss,speed_ms,0,blend_radius_m)
    movel([0.090387, -1.275971, -2.640734, -0.795684, 1.570796, 1.661183],accel_mss,speed_ms,0,blend_radius_m)
    movel([0.090598, -1.274287, -2.641682, -0.796420, 1.570796, 1.661394],accel_mss,speed_ms,0,blend_radius_m)
    movel([0.090772, -1.273008, -2.642399, -0.796982, 1.570796, 1.661569],accel_mss,speed_ms,0,blend_radius_m)
    movel([0.090933, -1.271977, -2.642976, -0.797436, 1.570796, 1.661730],accel_mss,speed_ms,0,blend_radius_m)
    movel([0.091081, -1.271125, -2.643452, -0.797812, 1.570796, 1.661878],accel_mss,speed_ms,0,blend_radius_m)
    movel([0.091342, -1.270867, -2.643595, -0.797926, 1.570796, 1.662139],accel_mss,speed_ms,0,blend_radius_m)
    movel([0.091673, -1.270956, -2.643546, -0.797887, 1.570796, 1.662469],accel_mss,speed_ms,0,blend_radius_m)
    movel([0.091927, -1.270981, -2.643532, -0.797876, 1.570796, 1.662723],accel_mss,speed_ms,0,blend_radius_m)
    movel([0.092311, -1.270967, -2.643540, -0.797882, 1.570796, 1.663108],accel_mss,speed_ms,0,blend_radius_m)
    movel([0.092453, -1.271196, -2.643412, -0.797781, 1.570796, 1.663250],accel_mss,speed_ms,0,blend_radius_m)
    movel([0.092461, -1.271755, -2.643100, -0.797534, 1.570796, 1.663257],accel_mss,speed_ms,0,blend_radius_m)
    movel([0.092320, -1.272984, -2.642413, -0.796993, 1.570796, 1.663116],accel_mss,speed_ms,0,blend_radius_m)
    movel([0.092175, -1.274267, -2.641693, -0.796429, 1.570796, 1.662971],accel_mss,speed_ms,0,blend_radius_m)
    movel([0.092201, -1.274815, -2.641385, -0.796189, 1.570796, 1.662997],accel_mss,speed_ms,0,blend_radius_m)
    movel([0.092385, -1.275020, -2.641269, -0.796099, 1.570796, 1.663181],accel_mss,speed_ms,0,blend_radius_m)
    movel([0.092744, -1.274999, -2.641281, -0.796109, 1.570796, 1.663541],accel_mss,speed_ms,0,blend_radius_m)
    movel([0.093158, -1.274747, -2.641423, -0.796219, 1.570796, 1.663954],accel_mss,speed_ms,0,blend_radius_m)
    movel([0.093440, -1.274359, -2.641641, -0.796389, 1.570796, 1.664237],accel_mss,speed_ms,0,blend_radius_m)
    movel([0.093651, -1.273687, -2.642019, -0.796684, 1.570796, 1.664448],accel_mss,speed_ms,0,blend_radius_m)
    movel([0.093890, -1.272343, -2.642771, -0.797275, 1.570796, 1.664686],accel_mss,speed_ms,0,blend_radius_m)
    movel([0.094066, -1.271271, -2.643370, -0.797748, 1.570796, 1.664863],accel_mss,speed_ms,0,blend_radius_m)
    movel([0.094187, -1.270730, -2.643672, -0.797987, 1.570796, 1.664983],accel_mss,speed_ms,0,blend_radius_m)
    movel([0.094304, -1.270407, -2.643852, -0.798130, 1.570796, 1.665100],accel_mss,speed_ms,0,blend_radius_m)
    movel([0.094576, -1.270134, -2.644004, -0.798251, 1.570796, 1.665372],accel_mss,speed_ms,0,blend_radius_m)
    movel([0.094860, -1.269922, -2.644122, -0.798345, 1.570796, 1.665657],accel_mss,speed_ms,0,blend_radius_m)
    movel([0.095215, -1.269546, -2.644331, -0.798512, 1.570796, 1.666012],accel_mss,speed_ms,0,blend_radius_m)
    movel([0.095415, -1.269125, -2.644565, -0.798699, 1.570796, 1.666211],accel_mss,speed_ms,0,blend_radius_m)
    movel([0.095501, -1.268757, -2.644769, -0.798863, 1.570796, 1.666298],accel_mss,speed_ms,0,blend_radius_m)
    movel([0.095460, -1.268527, -2.644896, -0.798965, 1.570796, 1.666256],accel_mss,speed_ms,0,blend_radius_m)
    movel([0.095278, -1.268390, -2.644972, -0.799026, 1.570796, 1.666075],accel_mss,speed_ms,0,blend_radius_m)
    movel([0.094918, -1.268325, -2.645008, -0.799055, 1.570796, 1.665714],accel_mss,speed_ms,0,blend_radius_m)
    movel([0.094621, -1.268149, -2.645106, -0.799134, 1.570796, 1.665417],accel_mss,speed_ms,0,blend_radius_m)
    movel([0.094596, -1.267894, -2.645247, -0.799247, 1.570796, 1.665392],accel_mss,speed_ms,0,blend_radius_m)
    movel([0.094629, -1.267268, -2.645594, -0.799527, 1.570796, 1.665426],accel_mss,speed_ms,0,blend_radius_m)
    movel([0.094635, -1.266534, -2.646000, -0.799855, 1.570796, 1.665432],accel_mss,speed_ms,0,blend_radius_m)
    movel([0.094510, -1.266152, -2.646210, -0.800026, 1.570796, 1.665306],accel_mss,speed_ms,0,blend_radius_m)
    movel([0.094243, -1.266052, -2.646266, -0.800071, 1.570796, 1.665039],accel_mss,speed_ms,0,blend_radius_m)
    movel([0.093835, -1.266187, -2.646191, -0.800011, 1.570796, 1.664631],accel_mss,speed_ms,0,blend_radius_m)
    movel([0.093555, -1.266396, -2.646076, -0.799917, 1.570796, 1.664352],accel_mss,speed_ms,0,blend_radius_m)
    movel([0.093224, -1.267045, -2.645717, -0.799627, 1.570796, 1.664020],accel_mss,speed_ms,0,blend_radius_m)
    movel([0.093066, -1.267765, -2.645319, -0.799305, 1.570796, 1.663862],accel_mss,speed_ms,0,blend_radius_m)
    movel([0.092919, -1.268403, -2.644965, -0.799020, 1.570796, 1.663715],accel_mss,speed_ms,0,blend_radius_m)
    movel([0.092764, -1.268768, -2.644763, -0.798858, 1.570796, 1.663561],accel_mss,speed_ms,0,blend_radius_m)
    movel([0.092248, -1.269162, -2.644544, -0.798683, 1.570796, 1.663044],accel_mss,speed_ms,0,blend_radius_m)
    movel([0.091948, -1.269335, -2.644448, -0.798606, 1.570796, 1.662744],accel_mss,speed_ms,0,blend_radius_m)
    movel([0.091695, -1.269594, -2.644304, -0.798491, 1.570796, 1.662491],accel_mss,speed_ms,0,blend_radius_m)
    movel([0.091391, -1.269862, -2.644155, -0.798372, 1.570796, 1.662187],accel_mss,speed_ms,0,blend_radius_m)
    movel([0.091166, -1.269655, -2.644270, -0.798464, 1.570796, 1.661962],accel_mss,speed_ms,0,blend_radius_m)
    movel([0.091445, -1.267615, -2.645402, -0.799372, 1.570796, 1.662241],accel_mss,speed_ms,0,blend_radius_m)
    movel([0.091760, -1.265579, -2.646526, -0.800284, 1.570796, 1.662556],accel_mss,speed_ms,0,blend_radius_m)
    movel([0.091988, -1.265169, -2.646752, -0.800468, 1.570796, 1.662785],accel_mss,speed_ms,0,blend_radius_m)
    movel([0.094110, -1.264369, -2.647192, -0.800828, 1.570796, 1.664907],accel_mss,speed_ms,0,blend_radius_m)
    movel([0.096668, -1.263512, -2.647663, -0.801215, 1.570796, 1.667464],accel_mss,speed_ms,0,blend_radius_m)
    movel([0.100580, -1.262238, -2.648361, -0.801791, 1.570796, 1.671376],accel_mss,speed_ms,0,blend_radius_m)
    movel([0.107027, -1.260177, -2.649485, -0.802727, 1.570796, 1.677824],accel_mss,speed_ms,0,blend_radius_m)
    movel([0.109986, -1.259263, -2.649982, -0.803144, 1.570796, 1.680783],accel_mss,speed_ms,0,blend_radius_m)
    movel([0.111807, -1.258730, -2.650271, -0.803388, 1.570796, 1.682603],accel_mss,speed_ms,0,blend_radius_m)
    movel([0.112142, -1.258735, -2.650269, -0.803386, 1.570796, 1.682938],accel_mss,speed_ms,0,blend_radius_m)
    movel([0.112198, -1.259199, -2.650016, -0.803173, 1.570796, 1.682994],accel_mss,speed_ms,0,blend_radius_m)
    movel([0.112144, -1.259741, -2.649722, -0.802926, 1.570796, 1.682940],accel_mss,speed_ms,0,blend_radius_m)
    movel([0.112026, -1.260556, -2.649279, -0.802555, 1.570796, 1.682822],accel_mss,speed_ms,0,blend_radius_m)
    movel([0.111880, -1.261504, -2.648761, -0.802124, 1.570796, 1.682676],accel_mss,speed_ms,0,blend_radius_m)
    speed_ms = 0.003
    movel([0.111880, -1.247359, -2.641944, -0.823086, 1.570796, 1.682676],accel_mss,speed_ms,0,blend_radius_m)
    speed_ms = 1.000
    movel([0.111880, -1.220520, -2.627929, -0.863940, 1.570796, 1.682676],accel_mss,speed_ms,0,blend_radius_m)
    movel([0.112627, -1.220290, -2.628048, -0.864051, 1.570796, 1.683424],accel_mss,speed_ms,0,blend_radius_m)
    movel([0.112627, -1.247131, -2.642066, -0.823192, 1.570796, 1.683424],accel_mss,speed_ms,0,blend_radius_m)
    speed_ms = 0.003
    movel([0.112627, -1.257695, -2.647192, -0.807502, 1.570796, 1.683424],accel_mss,speed_ms,0,blend_radius_m)
    speed_ms = 0.007
    movel([0.112348, -1.259448, -2.646239, -0.806702, 1.570796, 1.683144],accel_mss,speed_ms,0,blend_radius_m)
    movel([0.112042, -1.261409, -2.645167, -0.805813, 1.570796, 1.682838],accel_mss,speed_ms,0,blend_radius_m)
    movel([0.111746, -1.263319, -2.644120, -0.804950, 1.570796, 1.682543],accel_mss,speed_ms,0,blend_radius_m)
    movel([0.111426, -1.265348, -2.643001, -0.804039, 1.570796, 1.682222],accel_mss,speed_ms,0,blend_radius_m)
    movel([0.111175, -1.266791, -2.642204, -0.803395, 1.570796, 1.681972],accel_mss,speed_ms,0,blend_radius_m)
    movel([0.110968, -1.267885, -2.641596, -0.802907, 1.570796, 1.681765],accel_mss,speed_ms,0,blend_radius_m)
    movel([0.110743, -1.268207, -2.641418, -0.802765, 1.570796, 1.681539],accel_mss,speed_ms,0,blend_radius_m)
    movel([0.110333, -1.268397, -2.641312, -0.802680, 1.570796, 1.681130],accel_mss,speed_ms,0,blend_radius_m)
    movel([0.110030, -1.268480, -2.641266, -0.802643, 1.570796, 1.680827],accel_mss,speed_ms,0,blend_radius_m)
    movel([0.109555, -1.268608, -2.641194, -0.802586, 1.570796, 1.680351],accel_mss,speed_ms,0,blend_radius_m)
    movel([0.107397, -1.269273, -2.640824, -0.802292, 1.570796, 1.678193],accel_mss,speed_ms,0,blend_radius_m)
    movel([0.104864, -1.270064, -2.640383, -0.801942, 1.570796, 1.675660],accel_mss,speed_ms,0,blend_radius_m)
    movel([0.101985, -1.270976, -2.639874, -0.801539, 1.570796, 1.672782],accel_mss,speed_ms,0,blend_radius_m)
    movel([0.099128, -1.271889, -2.639363, -0.801137, 1.570796, 1.669925],accel_mss,speed_ms,0,blend_radius_m)
    movel([0.096668, -1.272675, -2.638922, -0.800792, 1.570796, 1.667465],accel_mss,speed_ms,0,blend_radius_m)
    movel([0.094528, -1.273355, -2.638540, -0.800494, 1.570796, 1.665324],accel_mss,speed_ms,0,blend_radius_m)
    movel([0.094023, -1.273494, -2.638462, -0.800433, 1.570796, 1.664820],accel_mss,speed_ms,0,blend_radius_m)
    movel([0.093394, -1.273693, -2.638350, -0.800346, 1.570796, 1.664191],accel_mss,speed_ms,0,blend_radius_m)
    movel([0.092643, -1.273938, -2.638212, -0.800239, 1.570796, 1.663439],accel_mss,speed_ms,0,blend_radius_m)
    movel([0.091820, -1.274214, -2.638057, -0.800118, 1.570796, 1.662617],accel_mss,speed_ms,0,blend_radius_m)
    movel([0.090138, -1.274763, -2.637747, -0.799879, 1.570796, 1.660934],accel_mss,speed_ms,0,blend_radius_m)
    movel([0.089596, -1.274814, -2.637719, -0.799857, 1.570796, 1.660392],accel_mss,speed_ms,0,blend_radius_m)
    movel([0.089396, -1.274569, -2.637857, -0.799963, 1.570796, 1.660192],accel_mss,speed_ms,0,blend_radius_m)
    movel([0.089475, -1.273808, -2.638285, -0.800296, 1.570796, 1.660272],accel_mss,speed_ms,0,blend_radius_m)
    movel([0.089572, -1.273233, -2.638609, -0.800547, 1.570796, 1.660368],accel_mss,speed_ms,0,blend_radius_m)
    movel([0.089807, -1.271526, -2.639566, -0.801297, 1.570796, 1.660604],accel_mss,speed_ms,0,blend_radius_m)
    movel([0.090080, -1.269491, -2.640703, -0.802195, 1.570796, 1.660876],accel_mss,speed_ms,0,blend_radius_m)
    movel([0.090372, -1.267236, -2.641957, -0.803196, 1.570796, 1.661168],accel_mss,speed_ms,0,blend_radius_m)
    movel([0.090752, -1.264317, -2.643570, -0.804501, 1.570796, 1.661548],accel_mss,speed_ms,0,blend_radius_m)
    movel([0.090996, -1.262630, -2.644498, -0.805261, 1.570796, 1.661793],accel_mss,speed_ms,0,blend_radius_m)
    movel([0.091188, -1.261486, -2.645125, -0.805778, 1.570796, 1.661985],accel_mss,speed_ms,0,blend_radius_m)
    movel([0.091578, -1.261046, -2.645366, -0.805977, 1.570796, 1.662374],accel_mss,speed_ms,0,blend_radius_m)
    movel([0.092647, -1.260652, -2.645581, -0.806155, 1.570796, 1.663443],accel_mss,speed_ms,0,blend_radius_m)
    movel([0.094365, -1.260061, -2.645904, -0.806424, 1.570796, 1.665162],accel_mss,speed_ms,0,blend_radius_m)
    movel([0.097839, -1.258925, -2.646524, -0.806941, 1.570796, 1.668635],accel_mss,speed_ms,0,blend_radius_m)
    movel([0.107546, -1.255806, -2.648216, -0.808367, 1.570796, 1.678343],accel_mss,speed_ms,0,blend_radius_m)
    movel([0.110803, -1.254792, -2.648763, -0.808834, 1.570796, 1.681599],accel_mss,speed_ms,0,blend_radius_m)
    movel([0.112623, -1.254251, -2.649055, -0.809083, 1.570796, 1.683419],accel_mss,speed_ms,0,blend_radius_m)
    movel([0.112969, -1.254257, -2.649052, -0.809080, 1.570796, 1.683766],accel_mss,speed_ms,0,blend_radius_m)
    movel([0.113078, -1.254715, -2.648805, -0.808869, 1.570796, 1.683875],accel_mss,speed_ms,0,blend_radius_m)
    movel([0.113013, -1.255305, -2.648487, -0.808598, 1.570796, 1.683809],accel_mss,speed_ms,0,blend_radius_m)
    movel([0.112812, -1.256551, -2.647812, -0.808025, 1.570796, 1.683609],accel_mss,speed_ms,0,blend_radius_m)
    movel([0.112627, -1.257695, -2.647192, -0.807502, 1.570796, 1.683424],accel_mss,speed_ms,0,blend_radius_m)
    speed_ms = 0.003
    movel([0.112627, -1.261278, -2.648885, -0.802226, 1.570796, 1.683424],accel_mss,speed_ms,0,blend_radius_m)
    speed_ms = 0.007
    movel([0.112348, -1.263027, -2.647928, -0.801433, 1.570796, 1.683144],accel_mss,speed_ms,0,blend_radius_m)
    movel([0.112042, -1.264984, -2.646854, -0.800551, 1.570796, 1.682838],accel_mss,speed_ms,0,blend_radius_m)
    movel([0.111746, -1.266891, -2.645803, -0.799696, 1.570796, 1.682543],accel_mss,speed_ms,0,blend_radius_m)
    movel([0.111426, -1.268916, -2.644681, -0.798792, 1.570796, 1.682222],accel_mss,speed_ms,0,blend_radius_m)
    movel([0.111175, -1.270356, -2.643881, -0.798153, 1.570796, 1.681972],accel_mss,speed_ms,0,blend_radius_m)
    movel([0.110968, -1.271448, -2.643271, -0.797670, 1.570796, 1.681765],accel_mss,speed_ms,0,blend_radius_m)
    movel([0.110743, -1.271769, -2.643092, -0.797528, 1.570796, 1.681539],accel_mss,speed_ms,0,blend_radius_m)
    movel([0.110333, -1.271958, -2.642986, -0.797444, 1.570796, 1.681130],accel_mss,speed_ms,0,blend_radius_m)
    movel([0.110030, -1.272041, -2.642940, -0.797408, 1.570796, 1.680827],accel_mss,speed_ms,0,blend_radius_m)
    movel([0.109555, -1.272170, -2.642868, -0.797351, 1.570796, 1.680351],accel_mss,speed_ms,0,blend_radius_m)
    movel([0.107397, -1.272833, -2.642497, -0.797059, 1.570796, 1.678193],accel_mss,speed_ms,0,blend_radius_m)
    movel([0.104864, -1.273622, -2.642055, -0.796712, 1.570796, 1.675660],accel_mss,speed_ms,0,blend_radius_m)
    movel([0.101985, -1.274533, -2.641544, -0.796313, 1.570796, 1.672782],accel_mss,speed_ms,0,blend_radius_m)
    movel([0.099128, -1.275444, -2.641031, -0.795914, 1.570796, 1.669925],accel_mss,speed_ms,0,blend_radius_m)
    movel([0.096668, -1.276228, -2.640589, -0.795572, 1.570796, 1.667465],accel_mss,speed_ms,0,blend_radius_m)
    movel([0.094528, -1.276907, -2.640206, -0.795277, 1.570796, 1.665324],accel_mss,speed_ms,0,blend_radius_m)
    movel([0.094023, -1.277045, -2.640127, -0.795216, 1.570796, 1.664820],accel_mss,speed_ms,0,blend_radius_m)
    movel([0.093394, -1.277243, -2.640015, -0.795130, 1.570796, 1.664191],accel_mss,speed_ms,0,blend_radius_m)
    movel([0.092643, -1.277489, -2.639877, -0.795024, 1.570796, 1.663439],accel_mss,speed_ms,0,blend_radius_m)
    movel([0.091820, -1.277764, -2.639721, -0.794904, 1.570796, 1.662617],accel_mss,speed_ms,0,blend_radius_m)
    movel([0.090138, -1.278312, -2.639411, -0.794667, 1.570796, 1.660934],accel_mss,speed_ms,0,blend_radius_m)
    movel([0.089596, -1.278362, -2.639382, -0.794645, 1.570796, 1.660392],accel_mss,speed_ms,0,blend_radius_m)
    movel([0.089396, -1.278118, -2.639520, -0.794751, 1.570796, 1.660192],accel_mss,speed_ms,0,blend_radius_m)
    movel([0.089475, -1.277358, -2.639950, -0.795080, 1.570796, 1.660272],accel_mss,speed_ms,0,blend_radius_m)
    movel([0.089572, -1.276785, -2.640275, -0.795330, 1.570796, 1.660368],accel_mss,speed_ms,0,blend_radius_m)
    movel([0.089807, -1.275081, -2.641235, -0.796073, 1.570796, 1.660604],accel_mss,speed_ms,0,blend_radius_m)
    movel([0.090080, -1.273050, -2.642375, -0.796963, 1.570796, 1.660876],accel_mss,speed_ms,0,blend_radius_m)
    movel([0.090372, -1.270800, -2.643633, -0.797956, 1.570796, 1.661168],accel_mss,speed_ms,0,blend_radius_m)
    movel([0.090752, -1.267887, -2.645251, -0.799250, 1.570796, 1.661548],accel_mss,speed_ms,0,blend_radius_m)
    movel([0.090996, -1.266203, -2.646182, -0.800004, 1.570796, 1.661793],accel_mss,speed_ms,0,blend_radius_m)
    movel([0.091188, -1.265061, -2.646811, -0.800516, 1.570796, 1.661985],accel_mss,speed_ms,0,blend_radius_m)
    movel([0.091578, -1.264622, -2.647053, -0.800714, 1.570796, 1.662374],accel_mss,speed_ms,0,blend_radius_m)
    movel([0.092647, -1.264229, -2.647269, -0.800891, 1.570796, 1.663443],accel_mss,speed_ms,0,blend_radius_m)
    movel([0.094365, -1.263639, -2.647593, -0.801157, 1.570796, 1.665162],accel_mss,speed_ms,0,blend_radius_m)
    movel([0.097839, -1.262505, -2.648214, -0.801670, 1.570796, 1.668635],accel_mss,speed_ms,0,blend_radius_m)
    movel([0.107546, -1.259392, -2.649911, -0.803085, 1.570796, 1.678343],accel_mss,speed_ms,0,blend_radius_m)
    movel([0.110803, -1.258380, -2.650461, -0.803548, 1.570796, 1.681599],accel_mss,speed_ms,0,blend_radius_m)
    movel([0.112623, -1.257840, -2.650754, -0.803795, 1.570796, 1.683419],accel_mss,speed_ms,0,blend_radius_m)
    movel([0.112969, -1.257846, -2.650750, -0.803793, 1.570796, 1.683766],accel_mss,speed_ms,0,blend_radius_m)
    movel([0.113078, -1.258304, -2.650502, -0.803583, 1.570796, 1.683875],accel_mss,speed_ms,0,blend_radius_m)
    movel([0.113013, -1.258892, -2.650183, -0.803314, 1.570796, 1.683809],accel_mss,speed_ms,0,blend_radius_m)
    movel([0.112812, -1.260136, -2.649507, -0.802746, 1.570796, 1.683609],accel_mss,speed_ms,0,blend_radius_m)
    movel([0.112627, -1.261278, -2.648885, -0.802226, 1.570796, 1.683424],accel_mss,speed_ms,0,blend_radius_m)
    speed_ms = 0.003
    movel([0.112627, -1.247131, -2.642066, -0.823192, 1.570796, 1.683424],accel_mss,speed_ms,0,blend_radius_m)
    speed_ms = 1.000
    movel([0.112627, -1.220290, -2.628048, -0.864051, 1.570796, 1.683424],accel_mss,speed_ms,0,blend_radius_m)
    movel([0.118475, -1.218867, -2.628781, -0.864741, 1.570796, 1.689271],accel_mss,speed_ms,0,blend_radius_m)
    movel([0.118475, -1.245724, -2.642817, -0.823848, 1.570796, 1.689271],accel_mss,speed_ms,0,blend_radius_m)
    speed_ms = 0.003
    movel([0.118475, -1.256295, -2.647951, -0.808143, 1.570796, 1.689271],accel_mss,speed_ms,0,blend_radius_m)
    speed_ms = 0.007
    movel([0.118642, -1.255906, -2.648162, -0.808321, 1.570796, 1.689439],accel_mss,speed_ms,0,blend_radius_m)
    movel([0.118971, -1.255659, -2.648295, -0.808435, 1.570796, 1.689767],accel_mss,speed_ms,0,blend_radius_m)
    movel([0.120090, -1.255250, -2.648516, -0.808623, 1.570796, 1.690887],accel_mss,speed_ms,0,blend_radius_m)
    movel([0.121216, -1.254877, -2.648717, -0.808794, 1.570796, 1.692013],accel_mss,speed_ms,0,blend_radius_m)
    movel([0.121456, -1.254929, -2.648689, -0.808771, 1.570796, 1.692252],accel_mss,speed_ms,0,blend_radius_m)
    movel([0.121429, -1.255682, -2.648283, -0.808424, 1.570796, 1.692226],accel_mss,speed_ms,0,blend_radius_m)
    movel([0.121359, -1.256453, -2.647866, -0.808070, 1.570796, 1.692155],accel_mss,speed_ms,0,blend_radius_m)
    movel([0.121264, -1.257344, -2.647383, -0.807662, 1.570796, 1.692060],accel_mss,speed_ms,0,blend_radius_m)
    movel([0.121103, -1.259178, -2.646386, -0.806825, 1.570796, 1.691900],accel_mss,speed_ms,0,blend_radius_m)
    movel([0.120972, -1.261800, -2.644953, -0.805636, 1.570796, 1.691768],accel_mss,speed_ms,0,blend_radius_m)
    movel([0.120868, -1.264596, -2.643416, -0.804376, 1.570796, 1.691665],accel_mss,speed_ms,0,blend_radius_m)
    movel([0.120965, -1.264813, -2.643297, -0.804279, 1.570796, 1.691761],accel_mss,speed_ms,0,blend_radius_m)
    movel([0.120902, -1.265202, -2.643082, -0.804105, 1.570796, 1.691698],accel_mss,speed_ms,0,blend_radius_m)
    movel([0.120470, -1.265588, -2.642869, -0.803932, 1.570796, 1.691266],accel_mss,speed_ms,0,blend_radius_m)
    movel([0.120082, -1.265788, -2.642759, -0.803843, 1.570796, 1.690879],accel_mss,speed_ms,0,blend_radius_m)
    movel([0.119727, -1.265906, -2.642693, -0.803790, 1.570796, 1.690524],accel_mss,speed_ms,0,blend_radius_m)
    movel([0.119381, -1.265588, -2.642869, -0.803932, 1.570796, 1.690177],accel_mss,speed_ms,0,blend_radius_m)
    movel([0.119064, -1.264014, -2.643737, -0.804638, 1.570796, 1.689860],accel_mss,speed_ms,0,blend_radius_m)
    movel([0.118772, -1.262381, -2.644635, -0.805373, 1.570796, 1.689568],accel_mss,speed_ms,0,blend_radius_m)
    movel([0.118582, -1.260960, -2.645413, -0.806016, 1.570796, 1.689378],accel_mss,speed_ms,0,blend_radius_m)
    movel([0.118465, -1.259399, -2.646265, -0.806725, 1.570796, 1.689261],accel_mss,speed_ms,0,blend_radius_m)
    movel([0.118440, -1.257782, -2.647145, -0.807462, 1.570796, 1.689236],accel_mss,speed_ms,0,blend_radius_m)
    movel([0.118475, -1.256295, -2.647951, -0.808143, 1.570796, 1.689271],accel_mss,speed_ms,0,blend_radius_m)
    speed_ms = 0.003
    movel([0.118475, -1.259880, -2.649646, -0.802862, 1.570796, 1.689271],accel_mss,speed_ms,0,blend_radius_m)
    speed_ms = 0.007
    movel([0.118642, -1.259492, -2.649857, -0.803040, 1.570796, 1.689439],accel_mss,speed_ms,0,blend_radius_m)
    movel([0.118971, -1.259245, -2.649991, -0.803152, 1.570796, 1.689767],accel_mss,speed_ms,0,blend_radius_m)
    movel([0.120090, -1.258837, -2.650213, -0.803339, 1.570796, 1.690887],accel_mss,speed_ms,0,blend_radius_m)
    movel([0.121216, -1.258466, -2.650415, -0.803509, 1.570796, 1.692013],accel_mss,speed_ms,0,blend_radius_m)
    movel([0.121456, -1.258517, -2.650387, -0.803485, 1.570796, 1.692252],accel_mss,speed_ms,0,blend_radius_m)
    movel([0.121429, -1.259268, -2.649979, -0.803142, 1.570796, 1.692226],accel_mss,speed_ms,0,blend_radius_m)
    movel([0.121359, -1.260038, -2.649560, -0.802791, 1.570796, 1.692155],accel_mss,speed_ms,0,blend_radius_m)
    movel([0.121264, -1.260927, -2.649076, -0.802386, 1.570796, 1.692060],accel_mss,speed_ms,0,blend_radius_m)
    movel([0.121103, -1.262758, -2.648076, -0.801555, 1.570796, 1.691900],accel_mss,speed_ms,0,blend_radius_m)
    movel([0.120972, -1.265375, -2.646639, -0.800375, 1.570796, 1.691768],accel_mss,speed_ms,0,blend_radius_m)
    movel([0.120868, -1.268165, -2.645097, -0.799126, 1.570796, 1.691665],accel_mss,speed_ms,0,blend_radius_m)
    movel([0.120965, -1.268381, -2.644977, -0.799030, 1.570796, 1.691761],accel_mss,speed_ms,0,blend_radius_m)
    movel([0.120902, -1.268770, -2.644762, -0.798857, 1.570796, 1.691698],accel_mss,speed_ms,0,blend_radius_m)
    movel([0.120470, -1.269155, -2.644548, -0.798686, 1.570796, 1.691266],accel_mss,speed_ms,0,blend_radius_m)
    movel([0.120082, -1.269355, -2.644437, -0.798597, 1.570796, 1.690879],accel_mss,speed_ms,0,blend_radius_m)
    movel([0.119727, -1.269472, -2.644372, -0.798545, 1.570796, 1.690524],accel_mss,speed_ms,0,blend_radius_m)
    movel([0.119381, -1.269155, -2.644548, -0.798686, 1.570796, 1.690177],accel_mss,speed_ms,0,blend_radius_m)
    movel([0.119064, -1.267584, -2.645419, -0.799386, 1.570796, 1.689860],accel_mss,speed_ms,0,blend_radius_m)
    movel([0.118772, -1.265954, -2.646319, -0.800115, 1.570796, 1.689568],accel_mss,speed_ms,0,blend_radius_m)
    movel([0.118582, -1.264536, -2.647100, -0.800753, 1.570796, 1.689378],accel_mss,speed_ms,0,blend_radius_m)
    movel([0.118465, -1.262979, -2.647955, -0.801455, 1.570796, 1.689261],accel_mss,speed_ms,0,blend_radius_m)
    movel([0.118440, -1.261365, -2.648837, -0.802187, 1.570796, 1.689236],accel_mss,speed_ms,0,blend_radius_m)
    movel([0.118475, -1.259880, -2.649646, -0.802862, 1.570796, 1.689271],accel_mss,speed_ms,0,blend_radius_m)
    speed_ms = 0.003
    movel([0.118475, -1.245724, -2.642817, -0.823848, 1.570796, 1.689271],accel_mss,speed_ms,0,blend_radius_m)
    speed_ms = 1.000
    movel([0.118475, -1.218867, -2.628781, -0.864741, 1.570796, 1.689271],accel_mss,speed_ms,0,blend_radius_m)
    movel([0.120041, -1.229230, -2.623391, -0.859768, 1.570796, 1.690837],accel_mss,speed_ms,0,blend_radius_m)
    movel([0.120041, -1.255970, -2.637290, -0.819128, 1.570796, 1.690837],accel_mss,speed_ms,0,blend_radius_m)
    speed_ms = 0.003
    movel([0.120041, -1.266486, -2.642372, -0.803531, 1.570796, 1.690837],accel_mss,speed_ms,0,blend_radius_m)
    speed_ms = 0.007
    movel([0.121226, -1.266003, -2.642639, -0.803746, 1.570796, 1.692023],accel_mss,speed_ms,0,blend_radius_m)
    movel([0.121974, -1.265746, -2.642781, -0.803861, 1.570796, 1.692771],accel_mss,speed_ms,0,blend_radius_m)
    movel([0.122521, -1.265587, -2.642869, -0.803932, 1.570796, 1.693317],accel_mss,speed_ms,0,blend_radius_m)
    movel([0.122965, -1.265496, -2.642920, -0.803973, 1.570796, 1.693761],accel_mss,speed_ms,0,blend_radius_m)
    movel([0.123374, -1.265460, -2.642940, -0.803989, 1.570796, 1.694171],accel_mss,speed_ms,0,blend_radius_m)
    movel([0.123869, -1.265479, -2.642929, -0.803981, 1.570796, 1.694665],accel_mss,speed_ms,0,blend_radius_m)
    movel([0.124152, -1.265567, -2.642881, -0.803942, 1.570796, 1.694948],accel_mss,speed_ms,0,blend_radius_m)
    movel([0.124317, -1.265756, -2.642776, -0.803857, 1.570796, 1.695114],accel_mss,speed_ms,0,blend_radius_m)
    movel([0.124415, -1.266094, -2.642589, -0.803706, 1.570796, 1.695212],accel_mss,speed_ms,0,blend_radius_m)
    movel([0.124415, -1.266769, -2.642216, -0.803404, 1.570796, 1.695211],accel_mss,speed_ms,0,blend_radius_m)
    movel([0.124075, -1.268942, -2.641009, -0.802438, 1.570796, 1.694871],accel_mss,speed_ms,0,blend_radius_m)
    movel([0.123687, -1.271228, -2.639733, -0.801428, 1.570796, 1.694483],accel_mss,speed_ms,0,blend_radius_m)
    movel([0.123510, -1.271587, -2.639532, -0.801270, 1.570796, 1.694306],accel_mss,speed_ms,0,blend_radius_m)
    movel([0.123023, -1.271869, -2.639374, -0.801146, 1.570796, 1.693820],accel_mss,speed_ms,0,blend_radius_m)
    movel([0.122565, -1.272067, -2.639263, -0.801059, 1.570796, 1.693361],accel_mss,speed_ms,0,blend_radius_m)
    movel([0.122004, -1.272280, -2.639143, -0.800965, 1.570796, 1.692800],accel_mss,speed_ms,0,blend_radius_m)
    movel([0.121262, -1.272566, -2.638983, -0.800840, 1.570796, 1.692059],accel_mss,speed_ms,0,blend_radius_m)
    movel([0.120728, -1.272809, -2.638847, -0.800733, 1.570796, 1.691524],accel_mss,speed_ms,0,blend_radius_m)
    movel([0.120243, -1.273086, -2.638691, -0.800612, 1.570796, 1.691039],accel_mss,speed_ms,0,blend_radius_m)
    movel([0.119665, -1.273472, -2.638474, -0.800443, 1.570796, 1.690461],accel_mss,speed_ms,0,blend_radius_m)
    movel([0.118666, -1.274175, -2.638079, -0.800135, 1.570796, 1.689463],accel_mss,speed_ms,0,blend_radius_m)
    movel([0.118375, -1.273980, -2.638188, -0.800221, 1.570796, 1.689171],accel_mss,speed_ms,0,blend_radius_m)
    movel([0.118029, -1.273614, -2.638394, -0.800381, 1.570796, 1.688826],accel_mss,speed_ms,0,blend_radius_m)
    movel([0.117532, -1.272666, -2.638927, -0.800796, 1.570796, 1.688329],accel_mss,speed_ms,0,blend_radius_m)
    movel([0.117085, -1.271656, -2.639493, -0.801240, 1.570796, 1.687881],accel_mss,speed_ms,0,blend_radius_m)
    movel([0.116878, -1.270903, -2.639915, -0.801571, 1.570796, 1.687675],accel_mss,speed_ms,0,blend_radius_m)
    movel([0.116838, -1.270587, -2.640091, -0.801711, 1.570796, 1.687634],accel_mss,speed_ms,0,blend_radius_m)
    movel([0.116822, -1.270209, -2.640302, -0.801878, 1.570796, 1.687618],accel_mss,speed_ms,0,blend_radius_m)
    movel([0.116822, -1.269830, -2.640514, -0.802045, 1.570796, 1.687618],accel_mss,speed_ms,0,blend_radius_m)
    movel([0.116849, -1.269514, -2.640690, -0.802185, 1.570796, 1.687646],accel_mss,speed_ms,0,blend_radius_m)
    movel([0.116920, -1.269100, -2.640921, -0.802368, 1.570796, 1.687716],accel_mss,speed_ms,0,blend_radius_m)
    movel([0.117181, -1.268584, -2.641208, -0.802597, 1.570796, 1.687977],accel_mss,speed_ms,0,blend_radius_m)
    movel([0.117494, -1.268230, -2.641405, -0.802754, 1.570796, 1.688291],accel_mss,speed_ms,0,blend_radius_m)
    movel([0.118205, -1.267582, -2.641765, -0.803042, 1.570796, 1.689001],accel_mss,speed_ms,0,blend_radius_m)
    movel([0.119043, -1.267008, -2.642083, -0.803298, 1.570796, 1.689839],accel_mss,speed_ms,0,blend_radius_m)
    movel([0.120041, -1.266486, -2.642372, -0.803531, 1.570796, 1.690837],accel_mss,speed_ms,0,blend_radius_m)
    speed_ms = 0.003
    movel([0.120041, -1.270052, -2.644050, -0.798288, 1.570796, 1.690837],accel_mss,speed_ms,0,blend_radius_m)
    speed_ms = 0.007
    movel([0.121226, -1.269570, -2.644318, -0.798502, 1.570796, 1.692023],accel_mss,speed_ms,0,blend_radius_m)
    movel([0.121974, -1.269313, -2.644460, -0.798615, 1.570796, 1.692771],accel_mss,speed_ms,0,blend_radius_m)
    movel([0.122521, -1.269154, -2.644549, -0.798686, 1.570796, 1.693317],accel_mss,speed_ms,0,blend_radius_m)
    movel([0.122965, -1.269063, -2.644599, -0.798727, 1.570796, 1.693761],accel_mss,speed_ms,0,blend_radius_m)
    movel([0.123374, -1.269028, -2.644619, -0.798742, 1.570796, 1.694171],accel_mss,speed_ms,0,blend_radius_m)
    movel([0.123869, -1.269047, -2.644608, -0.798734, 1.570796, 1.694665],accel_mss,speed_ms,0,blend_radius_m)
    movel([0.124152, -1.269134, -2.644560, -0.798695, 1.570796, 1.694948],accel_mss,speed_ms,0,blend_radius_m)
    movel([0.124317, -1.269323, -2.644455, -0.798611, 1.570796, 1.695114],accel_mss,speed_ms,0,blend_radius_m)
    movel([0.124415, -1.269660, -2.644268, -0.798461, 1.570796, 1.695212],accel_mss,speed_ms,0,blend_radius_m)
    movel([0.124415, -1.270334, -2.643893, -0.798162, 1.570796, 1.695211],accel_mss,speed_ms,0,blend_radius_m)
    movel([0.124075, -1.272502, -2.642682, -0.797204, 1.570796, 1.694871],accel_mss,speed_ms,0,blend_radius_m)
    movel([0.123687, -1.274784, -2.641402, -0.796203, 1.570796, 1.694483],accel_mss,speed_ms,0,blend_radius_m)
    movel([0.123510, -1.275142, -2.641201, -0.796046, 1.570796, 1.694306],accel_mss,speed_ms,0,blend_radius_m)
    movel([0.123023, -1.275424, -2.641042, -0.795923, 1.570796, 1.693820],accel_mss,speed_ms,0,blend_radius_m)
    movel([0.122565, -1.275621, -2.640931, -0.795837, 1.570796, 1.693361],accel_mss,speed_ms,0,blend_radius_m)
    movel([0.122004, -1.275834, -2.640811, -0.795744, 1.570796, 1.692800],accel_mss,speed_ms,0,blend_radius_m)
    movel([0.121262, -1.276120, -2.640650, -0.795619, 1.570796, 1.692059],accel_mss,speed_ms,0,blend_radius_m)
    movel([0.120728, -1.276361, -2.640514, -0.795514, 1.570796, 1.691524],accel_mss,speed_ms,0,blend_radius_m)
    movel([0.120243, -1.276639, -2.640357, -0.795393, 1.570796, 1.691039],accel_mss,speed_ms,0,blend_radius_m)
    movel([0.119665, -1.277024, -2.640140, -0.795226, 1.570796, 1.690461],accel_mss,speed_ms,0,blend_radius_m)
    movel([0.118666, -1.277725, -2.639743, -0.794921, 1.570796, 1.689463],accel_mss,speed_ms,0,blend_radius_m)
    movel([0.118375, -1.277530, -2.639853, -0.795006, 1.570796, 1.689171],accel_mss,speed_ms,0,blend_radius_m)
    movel([0.118029, -1.277165, -2.640060, -0.795164, 1.570796, 1.688826],accel_mss,speed_ms,0,blend_radius_m)
    movel([0.117532, -1.276219, -2.640594, -0.795576, 1.570796, 1.688329],accel_mss,speed_ms,0,blend_radius_m)
    movel([0.117085, -1.275211, -2.641162, -0.796016, 1.570796, 1.687881],accel_mss,speed_ms,0,blend_radius_m)
    movel([0.116878, -1.274460, -2.641585, -0.796345, 1.570796, 1.687675],accel_mss,speed_ms,0,blend_radius_m)
    movel([0.116838, -1.274144, -2.641762, -0.796483, 1.570796, 1.687634],accel_mss,speed_ms,0,blend_radius_m)
    movel([0.116822, -1.273767, -2.641974, -0.796648, 1.570796, 1.687618],accel_mss,speed_ms,0,blend_radius_m)
    movel([0.116822, -1.273389, -2.642185, -0.796814, 1.570796, 1.687618],accel_mss,speed_ms,0,blend_radius_m)
    movel([0.116849, -1.273073, -2.642362, -0.796953, 1.570796, 1.687646],accel_mss,speed_ms,0,blend_radius_m)
    movel([0.116920, -1.272660, -2.642594, -0.797135, 1.570796, 1.687716],accel_mss,speed_ms,0,blend_radius_m)
    movel([0.117181, -1.272145, -2.642882, -0.797362, 1.570796, 1.687977],accel_mss,speed_ms,0,blend_radius_m)
    movel([0.117494, -1.271792, -2.643079, -0.797518, 1.570796, 1.688291],accel_mss,speed_ms,0,blend_radius_m)
    movel([0.118205, -1.271145, -2.643440, -0.797803, 1.570796, 1.689001],accel_mss,speed_ms,0,blend_radius_m)
    movel([0.119043, -1.270573, -2.643760, -0.798057, 1.570796, 1.689839],accel_mss,speed_ms,0,blend_radius_m)
    movel([0.120041, -1.270052, -2.644050, -0.798288, 1.570796, 1.690837],accel_mss,speed_ms,0,blend_radius_m)
    speed_ms = 0.003
    movel([0.120041, -1.255970, -2.637290, -0.819128, 1.570796, 1.690837],accel_mss,speed_ms,0,blend_radius_m)
    speed_ms = 1.000
    movel([0.120041, -1.229230, -2.623391, -0.859768, 1.570796, 1.690837],accel_mss,speed_ms,0,blend_radius_m)
    movel([0.120623, -1.236312, -2.619637, -0.856440, 1.570796, 1.691420],accel_mss,speed_ms,0,blend_radius_m)
    movel([0.120623, -1.262968, -2.633444, -0.815978, 1.570796, 1.691420],accel_mss,speed_ms,0,blend_radius_m)
    speed_ms = 0.003
    movel([0.120623, -1.273444, -2.638490, -0.800455, 1.570796, 1.691420],accel_mss,speed_ms,0,blend_radius_m)
    speed_ms = 0.007
    movel([0.121538, -1.272993, -2.638744, -0.800653, 1.570796, 1.692335],accel_mss,speed_ms,0,blend_radius_m)
    movel([0.122479, -1.272594, -2.638967, -0.800827, 1.570796, 1.693276],accel_mss,speed_ms,0,blend_radius_m)
    movel([0.122911, -1.272555, -2.638989, -0.800845, 1.570796, 1.693707],accel_mss,speed_ms,0,blend_radius_m)
    movel([0.122366, -1.273226, -2.638613, -0.800551, 1.570796, 1.693163],accel_mss,speed_ms,0,blend_radius_m)
    movel([0.121831, -1.273575, -2.638416, -0.800398, 1.570796, 1.692627],accel_mss,speed_ms,0,blend_radius_m)
    movel([0.121074, -1.273981, -2.638188, -0.800220, 1.570796, 1.691871],accel_mss,speed_ms,0,blend_radius_m)
    movel([0.120299, -1.274351, -2.637980, -0.800059, 1.570796, 1.691095],accel_mss,speed_ms,0,blend_radius_m)
    movel([0.119690, -1.274584, -2.637848, -0.799957, 1.570796, 1.690487],accel_mss,speed_ms,0,blend_radius_m)
    movel([0.119386, -1.274630, -2.637822, -0.799937, 1.570796, 1.690183],accel_mss,speed_ms,0,blend_radius_m)
    movel([0.119481, -1.274207, -2.638061, -0.800122, 1.570796, 1.690277],accel_mss,speed_ms,0,blend_radius_m)
    movel([0.119937, -1.273855, -2.638259, -0.800275, 1.570796, 1.690733],accel_mss,speed_ms,0,blend_radius_m)
    movel([0.120623, -1.273444, -2.638490, -0.800455, 1.570796, 1.691420],accel_mss,speed_ms,0,blend_radius_m)
    speed_ms = 0.003
    movel([0.120623, -1.276996, -2.640155, -0.795238, 1.570796, 1.691420],accel_mss,speed_ms,0,blend_radius_m)
    speed_ms = 0.007
    movel([0.121538, -1.276545, -2.640410, -0.795434, 1.570796, 1.692335],accel_mss,speed_ms,0,blend_radius_m)
    movel([0.122479, -1.276148, -2.640634, -0.795607, 1.570796, 1.693276],accel_mss,speed_ms,0,blend_radius_m)
    movel([0.122911, -1.276108, -2.640656, -0.795624, 1.570796, 1.693707],accel_mss,speed_ms,0,blend_radius_m)
    movel([0.122366, -1.276778, -2.640279, -0.795333, 1.570796, 1.693163],accel_mss,speed_ms,0,blend_radius_m)
    movel([0.121831, -1.277126, -2.640082, -0.795181, 1.570796, 1.692627],accel_mss,speed_ms,0,blend_radius_m)
    movel([0.121074, -1.277531, -2.639853, -0.795005, 1.570796, 1.691871],accel_mss,speed_ms,0,blend_radius_m)
    movel([0.120299, -1.277900, -2.639644, -0.794845, 1.570796, 1.691095],accel_mss,speed_ms,0,blend_radius_m)
    movel([0.119690, -1.278133, -2.639512, -0.794744, 1.570796, 1.690487],accel_mss,speed_ms,0,blend_radius_m)
    movel([0.119386, -1.278179, -2.639486, -0.794724, 1.570796, 1.690183],accel_mss,speed_ms,0,blend_radius_m)
    movel([0.119481, -1.277757, -2.639725, -0.794907, 1.570796, 1.690277],accel_mss,speed_ms,0,blend_radius_m)
    movel([0.119937, -1.277406, -2.639924, -0.795060, 1.570796, 1.690733],accel_mss,speed_ms,0,blend_radius_m)
    movel([0.120623, -1.276996, -2.640155, -0.795238, 1.570796, 1.691420],accel_mss,speed_ms,0,blend_radius_m)
    speed_ms = 0.003
    movel([0.120623, -1.262968, -2.633444, -0.815978, 1.570796, 1.691420],accel_mss,speed_ms,0,blend_radius_m)
    speed_ms = 1.000
    movel([0.120623, -1.236312, -2.619637, -0.856440, 1.570796, 1.691420],accel_mss,speed_ms,0,blend_radius_m)
    movel([0.120709, -1.237636, -2.618929, -0.855824, 1.570796, 1.691505],accel_mss,speed_ms,0,blend_radius_m)
    movel([0.120709, -1.264276, -2.632718, -0.815395, 1.570796, 1.691505],accel_mss,speed_ms,0,blend_radius_m)
    speed_ms = 0.003
    movel([0.120709, -1.274745, -2.637757, -0.799887, 1.570796, 1.691505],accel_mss,speed_ms,0,blend_radius_m)
    speed_ms = 0.007
    movel([0.121089, -1.274555, -2.637864, -0.799969, 1.570796, 1.691885],accel_mss,speed_ms,0,blend_radius_m)
    movel([0.121512, -1.274333, -2.637990, -0.800067, 1.570796, 1.692308],accel_mss,speed_ms,0,blend_radius_m)
    movel([0.121915, -1.274114, -2.638113, -0.800162, 1.570796, 1.692711],accel_mss,speed_ms,0,blend_radius_m)
    movel([0.122224, -1.273935, -2.638214, -0.800240, 1.570796, 1.693020],accel_mss,speed_ms,0,blend_radius_m)
    movel([0.122594, -1.273721, -2.638334, -0.800334, 1.570796, 1.693390],accel_mss,speed_ms,0,blend_radius_m)
    movel([0.122927, -1.273623, -2.638389, -0.800377, 1.570796, 1.693724],accel_mss,speed_ms,0,blend_radius_m)
    movel([0.123154, -1.273808, -2.638285, -0.800296, 1.570796, 1.693950],accel_mss,speed_ms,0,blend_radius_m)
    movel([0.122937, -1.274126, -2.638106, -0.800157, 1.570796, 1.693733],accel_mss,speed_ms,0,blend_radius_m)
    movel([0.122394, -1.274377, -2.637965, -0.800047, 1.570796, 1.693190],accel_mss,speed_ms,0,blend_radius_m)
    movel([0.122493, -1.274583, -2.637849, -0.799957, 1.570796, 1.693289],accel_mss,speed_ms,0,blend_radius_m)
    movel([0.122823, -1.274541, -2.637872, -0.799975, 1.570796, 1.693620],accel_mss,speed_ms,0,blend_radius_m)
    movel([0.123129, -1.274442, -2.637928, -0.800019, 1.570796, 1.693926],accel_mss,speed_ms,0,blend_radius_m)
    movel([0.123433, -1.274098, -2.638122, -0.800169, 1.570796, 1.694230],accel_mss,speed_ms,0,blend_radius_m)
    movel([0.123760, -1.273889, -2.638239, -0.800260, 1.570796, 1.694556],accel_mss,speed_ms,0,blend_radius_m)
    movel([0.124094, -1.273901, -2.638233, -0.800255, 1.570796, 1.694890],accel_mss,speed_ms,0,blend_radius_m)
    movel([0.124564, -1.273889, -2.638239, -0.800260, 1.570796, 1.695360],accel_mss,speed_ms,0,blend_radius_m)
    movel([0.125059, -1.273833, -2.638271, -0.800285, 1.570796, 1.695855],accel_mss,speed_ms,0,blend_radius_m)
    movel([0.125372, -1.273722, -2.638333, -0.800333, 1.570796, 1.696168],accel_mss,speed_ms,0,blend_radius_m)
    movel([0.125657, -1.273693, -2.638350, -0.800346, 1.570796, 1.696454],accel_mss,speed_ms,0,blend_radius_m)
    movel([0.125972, -1.273513, -2.638451, -0.800425, 1.570796, 1.696768],accel_mss,speed_ms,0,blend_radius_m)
    movel([0.126196, -1.273572, -2.638418, -0.800399, 1.570796, 1.696993],accel_mss,speed_ms,0,blend_radius_m)
    movel([0.126436, -1.273622, -2.638390, -0.800377, 1.570796, 1.697232],accel_mss,speed_ms,0,blend_radius_m)
    movel([0.126810, -1.273519, -2.638448, -0.800422, 1.570796, 1.697606],accel_mss,speed_ms,0,blend_radius_m)
    movel([0.127277, -1.273338, -2.638550, -0.800501, 1.570796, 1.698073],accel_mss,speed_ms,0,blend_radius_m)
    movel([0.127645, -1.273239, -2.638605, -0.800545, 1.570796, 1.698441],accel_mss,speed_ms,0,blend_radius_m)
    movel([0.128058, -1.273284, -2.638580, -0.800525, 1.570796, 1.698854],accel_mss,speed_ms,0,blend_radius_m)
    movel([0.128268, -1.273441, -2.638492, -0.800456, 1.570796, 1.699064],accel_mss,speed_ms,0,blend_radius_m)
    movel([0.128442, -1.273661, -2.638368, -0.800360, 1.570796, 1.699239],accel_mss,speed_ms,0,blend_radius_m)
    movel([0.128502, -1.273887, -2.638241, -0.800261, 1.570796, 1.699298],accel_mss,speed_ms,0,blend_radius_m)
    movel([0.128278, -1.274189, -2.638071, -0.800129, 1.570796, 1.699074],accel_mss,speed_ms,0,blend_radius_m)
    movel([0.128301, -1.274481, -2.637906, -0.800002, 1.570796, 1.699097],accel_mss,speed_ms,0,blend_radius_m)
    movel([0.128456, -1.274704, -2.637781, -0.799905, 1.570796, 1.699252],accel_mss,speed_ms,0,blend_radius_m)
    movel([0.128142, -1.275293, -2.637448, -0.799648, 1.570796, 1.698939],accel_mss,speed_ms,0,blend_radius_m)
    movel([0.127643, -1.275903, -2.637103, -0.799382, 1.570796, 1.698439],accel_mss,speed_ms,0,blend_radius_m)
    movel([0.127331, -1.276274, -2.636894, -0.799221, 1.570796, 1.698128],accel_mss,speed_ms,0,blend_radius_m)
    movel([0.127066, -1.276603, -2.636708, -0.799078, 1.570796, 1.697863],accel_mss,speed_ms,0,blend_radius_m)
    movel([0.126852, -1.276880, -2.636551, -0.798958, 1.570796, 1.697648],accel_mss,speed_ms,0,blend_radius_m)
    movel([0.126937, -1.277097, -2.636428, -0.798864, 1.570796, 1.697734],accel_mss,speed_ms,0,blend_radius_m)
    movel([0.127240, -1.277322, -2.636300, -0.798767, 1.570796, 1.698036],accel_mss,speed_ms,0,blend_radius_m)
    movel([0.127528, -1.277565, -2.636162, -0.798662, 1.570796, 1.698325],accel_mss,speed_ms,0,blend_radius_m)
    movel([0.127643, -1.277822, -2.636017, -0.798551, 1.570796, 1.698439],accel_mss,speed_ms,0,blend_radius_m)
    movel([0.127335, -1.278017, -2.635906, -0.798466, 1.570796, 1.698131],accel_mss,speed_ms,0,blend_radius_m)
    movel([0.127124, -1.277913, -2.635965, -0.798511, 1.570796, 1.697920],accel_mss,speed_ms,0,blend_radius_m)
    movel([0.126991, -1.277725, -2.636071, -0.798592, 1.570796, 1.697788],accel_mss,speed_ms,0,blend_radius_m)
    movel([0.126865, -1.277536, -2.636179, -0.798674, 1.570796, 1.697661],accel_mss,speed_ms,0,blend_radius_m)
    movel([0.126558, -1.277649, -2.636115, -0.798625, 1.570796, 1.697354],accel_mss,speed_ms,0,blend_radius_m)
    movel([0.126435, -1.277451, -2.636227, -0.798711, 1.570796, 1.697231],accel_mss,speed_ms,0,blend_radius_m)
    movel([0.126185, -1.277352, -2.636283, -0.798754, 1.570796, 1.696981],accel_mss,speed_ms,0,blend_radius_m)
    movel([0.126273, -1.277071, -2.636443, -0.798876, 1.570796, 1.697069],accel_mss,speed_ms,0,blend_radius_m)
    movel([0.126374, -1.276773, -2.636611, -0.799004, 1.570796, 1.697170],accel_mss,speed_ms,0,blend_radius_m)
    movel([0.126672, -1.276609, -2.636704, -0.799076, 1.570796, 1.697468],accel_mss,speed_ms,0,blend_radius_m)
    movel([0.126485, -1.276461, -2.636788, -0.799140, 1.570796, 1.697281],accel_mss,speed_ms,0,blend_radius_m)
    movel([0.126217, -1.276701, -2.636652, -0.799036, 1.570796, 1.697013],accel_mss,speed_ms,0,blend_radius_m)
    movel([0.125927, -1.276921, -2.636528, -0.798941, 1.570796, 1.696723],accel_mss,speed_ms,0,blend_radius_m)
    movel([0.125642, -1.277168, -2.636387, -0.798833, 1.570796, 1.696438],accel_mss,speed_ms,0,blend_radius_m)
    movel([0.125248, -1.277363, -2.636277, -0.798749, 1.570796, 1.696044],accel_mss,speed_ms,0,blend_radius_m)
    movel([0.124945, -1.277567, -2.636161, -0.798661, 1.570796, 1.695741],accel_mss,speed_ms,0,blend_radius_m)
    movel([0.124618, -1.277726, -2.636071, -0.798592, 1.570796, 1.695414],accel_mss,speed_ms,0,blend_radius_m)
    movel([0.124820, -1.277864, -2.635992, -0.798532, 1.570796, 1.695616],accel_mss,speed_ms,0,blend_radius_m)
    movel([0.125120, -1.277761, -2.636051, -0.798577, 1.570796, 1.695916],accel_mss,speed_ms,0,blend_radius_m)
    movel([0.125422, -1.277761, -2.636051, -0.798577, 1.570796, 1.696218],accel_mss,speed_ms,0,blend_radius_m)
    movel([0.125734, -1.277782, -2.636039, -0.798568, 1.570796, 1.696530],accel_mss,speed_ms,0,blend_radius_m)
    movel([0.125551, -1.277664, -2.636106, -0.798619, 1.570796, 1.696347],accel_mss,speed_ms,0,blend_radius_m)
    movel([0.125887, -1.277557, -2.636167, -0.798665, 1.570796, 1.696683],accel_mss,speed_ms,0,blend_radius_m)
    movel([0.126035, -1.277708, -2.636081, -0.798600, 1.570796, 1.696831],accel_mss,speed_ms,0,blend_radius_m)
    movel([0.126335, -1.277740, -2.636063, -0.798586, 1.570796, 1.697131],accel_mss,speed_ms,0,blend_radius_m)
    movel([0.126542, -1.277914, -2.635964, -0.798511, 1.570796, 1.697338],accel_mss,speed_ms,0,blend_radius_m)
    movel([0.126874, -1.277969, -2.635933, -0.798487, 1.570796, 1.697670],accel_mss,speed_ms,0,blend_radius_m)
    movel([0.127085, -1.278190, -2.635807, -0.798391, 1.570796, 1.697881],accel_mss,speed_ms,0,blend_radius_m)
    movel([0.126908, -1.278486, -2.635639, -0.798264, 1.570796, 1.697705],accel_mss,speed_ms,0,blend_radius_m)
    movel([0.126872, -1.278838, -2.635439, -0.798112, 1.570796, 1.697668],accel_mss,speed_ms,0,blend_radius_m)
    movel([0.126732, -1.279107, -2.635286, -0.797996, 1.570796, 1.697528],accel_mss,speed_ms,0,blend_radius_m)
    movel([0.127032, -1.278943, -2.635379, -0.798067, 1.570796, 1.697828],accel_mss,speed_ms,0,blend_radius_m)
    movel([0.127020, -1.278551, -2.635602, -0.798236, 1.570796, 1.697816],accel_mss,speed_ms,0,blend_radius_m)
    movel([0.127207, -1.278254, -2.635771, -0.798364, 1.570796, 1.698004],accel_mss,speed_ms,0,blend_radius_m)
    movel([0.127325, -1.278449, -2.635660, -0.798280, 1.570796, 1.698121],accel_mss,speed_ms,0,blend_radius_m)
    movel([0.127108, -1.278786, -2.635469, -0.798134, 1.570796, 1.697904],accel_mss,speed_ms,0,blend_radius_m)
    movel([0.127401, -1.278693, -2.635522, -0.798175, 1.570796, 1.698197],accel_mss,speed_ms,0,blend_radius_m)
    movel([0.127190, -1.279254, -2.635202, -0.797933, 1.570796, 1.697986],accel_mss,speed_ms,0,blend_radius_m)
    movel([0.126973, -1.279513, -2.635055, -0.797821, 1.570796, 1.697769],accel_mss,speed_ms,0,blend_radius_m)
    movel([0.126665, -1.279694, -2.634952, -0.797744, 1.570796, 1.697462],accel_mss,speed_ms,0,blend_radius_m)
    movel([0.126509, -1.280002, -2.634776, -0.797611, 1.570796, 1.697305],accel_mss,speed_ms,0,blend_radius_m)
    movel([0.126164, -1.280432, -2.634530, -0.797426, 1.570796, 1.696960],accel_mss,speed_ms,0,blend_radius_m)
    movel([0.125846, -1.280805, -2.634317, -0.797267, 1.570796, 1.696642],accel_mss,speed_ms,0,blend_radius_m)
    movel([0.126192, -1.280881, -2.634274, -0.797234, 1.570796, 1.696988],accel_mss,speed_ms,0,blend_radius_m)
    movel([0.126470, -1.281020, -2.634194, -0.797174, 1.570796, 1.697267],accel_mss,speed_ms,0,blend_radius_m)
    movel([0.126536, -1.281240, -2.634069, -0.797080, 1.570796, 1.697332],accel_mss,speed_ms,0,blend_radius_m)
    movel([0.126661, -1.281453, -2.633947, -0.796989, 1.570796, 1.697458],accel_mss,speed_ms,0,blend_radius_m)
    movel([0.126532, -1.281783, -2.633758, -0.796848, 1.570796, 1.697328],accel_mss,speed_ms,0,blend_radius_m)
    movel([0.126278, -1.282138, -2.633555, -0.796697, 1.570796, 1.697074],accel_mss,speed_ms,0,blend_radius_m)
    movel([0.125958, -1.282547, -2.633320, -0.796522, 1.570796, 1.696754],accel_mss,speed_ms,0,blend_radius_m)
    movel([0.125587, -1.282807, -2.633171, -0.796411, 1.570796, 1.696383],accel_mss,speed_ms,0,blend_radius_m)
    movel([0.125858, -1.282592, -2.633294, -0.796503, 1.570796, 1.696654],accel_mss,speed_ms,0,blend_radius_m)
    movel([0.125869, -1.282306, -2.633458, -0.796625, 1.570796, 1.696665],accel_mss,speed_ms,0,blend_radius_m)
    movel([0.126028, -1.282007, -2.633629, -0.796752, 1.570796, 1.696825],accel_mss,speed_ms,0,blend_radius_m)
    movel([0.126232, -1.281491, -2.633925, -0.796973, 1.570796, 1.697029],accel_mss,speed_ms,0,blend_radius_m)
    movel([0.126003, -1.281427, -2.633962, -0.797000, 1.570796, 1.696799],accel_mss,speed_ms,0,blend_radius_m)
    movel([0.125957, -1.281160, -2.634114, -0.797114, 1.570796, 1.696753],accel_mss,speed_ms,0,blend_radius_m)
    movel([0.125809, -1.281008, -2.634201, -0.797180, 1.570796, 1.696605],accel_mss,speed_ms,0,blend_radius_m)
    movel([0.125586, -1.280893, -2.634267, -0.797229, 1.570796, 1.696383],accel_mss,speed_ms,0,blend_radius_m)
    movel([0.125377, -1.280815, -2.634312, -0.797262, 1.570796, 1.696173],accel_mss,speed_ms,0,blend_radius_m)
    movel([0.125610, -1.280532, -2.634473, -0.797384, 1.570796, 1.696406],accel_mss,speed_ms,0,blend_radius_m)
    movel([0.125992, -1.280122, -2.634708, -0.797560, 1.570796, 1.696789],accel_mss,speed_ms,0,blend_radius_m)
    movel([0.126321, -1.279769, -2.634909, -0.797711, 1.570796, 1.697118],accel_mss,speed_ms,0,blend_radius_m)
    movel([0.126533, -1.279429, -2.635102, -0.797857, 1.570796, 1.697330],accel_mss,speed_ms,0,blend_radius_m)
    movel([0.126193, -1.279649, -2.634977, -0.797763, 1.570796, 1.696989],accel_mss,speed_ms,0,blend_radius_m)
    movel([0.125766, -1.280010, -2.634771, -0.797608, 1.570796, 1.696563],accel_mss,speed_ms,0,blend_radius_m)
    movel([0.125446, -1.280382, -2.634559, -0.797448, 1.570796, 1.696242],accel_mss,speed_ms,0,blend_radius_m)
    movel([0.125139, -1.280519, -2.634481, -0.797389, 1.570796, 1.695935],accel_mss,speed_ms,0,blend_radius_m)
    movel([0.124558, -1.280955, -2.634232, -0.797203, 1.570796, 1.695354],accel_mss,speed_ms,0,blend_radius_m)
    movel([0.124536, -1.281261, -2.634056, -0.797071, 1.570796, 1.695333],accel_mss,speed_ms,0,blend_radius_m)
    movel([0.124872, -1.281302, -2.634033, -0.797054, 1.570796, 1.695668],accel_mss,speed_ms,0,blend_radius_m)
    movel([0.125134, -1.281286, -2.634043, -0.797061, 1.570796, 1.695931],accel_mss,speed_ms,0,blend_radius_m)
    movel([0.125420, -1.281158, -2.634116, -0.797116, 1.570796, 1.696217],accel_mss,speed_ms,0,blend_radius_m)
    movel([0.125608, -1.281312, -2.634027, -0.797049, 1.570796, 1.696404],accel_mss,speed_ms,0,blend_radius_m)
    movel([0.125786, -1.281536, -2.633900, -0.796954, 1.570796, 1.696583],accel_mss,speed_ms,0,blend_radius_m)
    movel([0.125996, -1.281628, -2.633847, -0.796914, 1.570796, 1.696792],accel_mss,speed_ms,0,blend_radius_m)
    movel([0.125747, -1.282027, -2.633618, -0.796744, 1.570796, 1.696543],accel_mss,speed_ms,0,blend_radius_m)
    movel([0.125404, -1.282465, -2.633367, -0.796557, 1.570796, 1.696200],accel_mss,speed_ms,0,blend_radius_m)
    movel([0.125296, -1.282737, -2.633211, -0.796441, 1.570796, 1.696093],accel_mss,speed_ms,0,blend_radius_m)
    movel([0.124953, -1.283047, -2.633033, -0.796309, 1.570796, 1.695749],accel_mss,speed_ms,0,blend_radius_m)
    movel([0.124458, -1.283370, -2.632848, -0.796172, 1.570796, 1.695255],accel_mss,speed_ms,0,blend_radius_m)
    movel([0.123806, -1.283823, -2.632587, -0.795979, 1.570796, 1.694603],accel_mss,speed_ms,0,blend_radius_m)
    movel([0.124318, -1.283650, -2.632687, -0.796053, 1.570796, 1.695114],accel_mss,speed_ms,0,blend_radius_m)
    movel([0.124661, -1.283507, -2.632769, -0.796113, 1.570796, 1.695458],accel_mss,speed_ms,0,blend_radius_m)
    movel([0.124937, -1.283298, -2.632889, -0.796202, 1.570796, 1.695733],accel_mss,speed_ms,0,blend_radius_m)
    movel([0.125165, -1.283024, -2.633046, -0.796319, 1.570796, 1.695962],accel_mss,speed_ms,0,blend_radius_m)
    movel([0.125011, -1.283420, -2.632819, -0.796150, 1.570796, 1.695807],accel_mss,speed_ms,0,blend_radius_m)
    movel([0.124648, -1.283719, -2.632647, -0.796023, 1.570796, 1.695444],accel_mss,speed_ms,0,blend_radius_m)
    movel([0.124301, -1.283928, -2.632527, -0.795935, 1.570796, 1.695097],accel_mss,speed_ms,0,blend_radius_m)
    movel([0.123990, -1.284200, -2.632370, -0.795819, 1.570796, 1.694786],accel_mss,speed_ms,0,blend_radius_m)
    movel([0.123623, -1.284184, -2.632379, -0.795826, 1.570796, 1.694419],accel_mss,speed_ms,0,blend_radius_m)
    movel([0.123370, -1.284155, -2.632396, -0.795838, 1.570796, 1.694166],accel_mss,speed_ms,0,blend_radius_m)
    movel([0.122926, -1.284478, -2.632210, -0.795701, 1.570796, 1.693723],accel_mss,speed_ms,0,blend_radius_m)
    movel([0.122673, -1.284726, -2.632067, -0.795596, 1.570796, 1.693469],accel_mss,speed_ms,0,blend_radius_m)
    movel([0.122307, -1.284621, -2.632128, -0.795641, 1.570796, 1.693104],accel_mss,speed_ms,0,blend_radius_m)
    movel([0.122004, -1.284684, -2.632091, -0.795614, 1.570796, 1.692801],accel_mss,speed_ms,0,blend_radius_m)
    movel([0.121661, -1.284967, -2.631928, -0.795494, 1.570796, 1.692457],accel_mss,speed_ms,0,blend_radius_m)
    movel([0.121351, -1.285158, -2.631818, -0.795413, 1.570796, 1.692148],accel_mss,speed_ms,0,blend_radius_m)
    movel([0.121025, -1.285375, -2.631693, -0.795321, 1.570796, 1.691821],accel_mss,speed_ms,0,blend_radius_m)
    movel([0.120795, -1.285611, -2.631557, -0.795222, 1.570796, 1.691591],accel_mss,speed_ms,0,blend_radius_m)
    movel([0.120927, -1.285305, -2.631733, -0.795351, 1.570796, 1.691724],accel_mss,speed_ms,0,blend_radius_m)
    movel([0.120541, -1.285236, -2.631773, -0.795380, 1.570796, 1.691337],accel_mss,speed_ms,0,blend_radius_m)
    movel([0.120155, -1.285378, -2.631691, -0.795320, 1.570796, 1.690951],accel_mss,speed_ms,0,blend_radius_m)
    movel([0.119775, -1.285519, -2.631609, -0.795260, 1.570796, 1.690571],accel_mss,speed_ms,0,blend_radius_m)
    movel([0.119308, -1.285630, -2.631546, -0.795214, 1.570796, 1.690104],accel_mss,speed_ms,0,blend_radius_m)
    movel([0.119086, -1.285504, -2.631618, -0.795267, 1.570796, 1.689882],accel_mss,speed_ms,0,blend_radius_m)
    movel([0.118778, -1.285404, -2.631676, -0.795309, 1.570796, 1.689574],accel_mss,speed_ms,0,blend_radius_m)
    movel([0.118635, -1.285235, -2.631773, -0.795381, 1.570796, 1.689431],accel_mss,speed_ms,0,blend_radius_m)
    movel([0.118460, -1.285035, -2.631889, -0.795465, 1.570796, 1.689257],accel_mss,speed_ms,0,blend_radius_m)
    movel([0.118223, -1.284987, -2.631916, -0.795485, 1.570796, 1.689019],accel_mss,speed_ms,0,blend_radius_m)
    movel([0.118344, -1.285324, -2.631722, -0.795343, 1.570796, 1.689141],accel_mss,speed_ms,0,blend_radius_m)
    movel([0.118538, -1.285556, -2.631588, -0.795245, 1.570796, 1.689335],accel_mss,speed_ms,0,blend_radius_m)
    movel([0.118550, -1.285829, -2.631430, -0.795130, 1.570796, 1.689347],accel_mss,speed_ms,0,blend_radius_m)
    movel([0.118849, -1.285637, -2.631542, -0.795211, 1.570796, 1.689645],accel_mss,speed_ms,0,blend_radius_m)
    movel([0.118996, -1.285840, -2.631424, -0.795125, 1.570796, 1.689792],accel_mss,speed_ms,0,blend_radius_m)
    movel([0.118698, -1.286006, -2.631328, -0.795055, 1.570796, 1.689495],accel_mss,speed_ms,0,blend_radius_m)
    movel([0.118450, -1.285983, -2.631341, -0.795064, 1.570796, 1.689246],accel_mss,speed_ms,0,blend_radius_m)
    movel([0.118230, -1.285882, -2.631400, -0.795107, 1.570796, 1.689027],accel_mss,speed_ms,0,blend_radius_m)
    movel([0.118043, -1.285700, -2.631505, -0.795184, 1.570796, 1.688839],accel_mss,speed_ms,0,blend_radius_m)
    movel([0.117955, -1.285495, -2.631623, -0.795271, 1.570796, 1.688751],accel_mss,speed_ms,0,blend_radius_m)
    movel([0.118003, -1.285194, -2.631797, -0.795398, 1.570796, 1.688799],accel_mss,speed_ms,0,blend_radius_m)
    movel([0.118007, -1.284913, -2.631959, -0.795517, 1.570796, 1.688804],accel_mss,speed_ms,0,blend_radius_m)
    movel([0.118087, -1.284517, -2.632187, -0.795684, 1.570796, 1.688883],accel_mss,speed_ms,0,blend_radius_m)
    movel([0.118058, -1.284204, -2.632368, -0.795817, 1.570796, 1.688855],accel_mss,speed_ms,0,blend_radius_m)
    movel([0.117873, -1.283980, -2.632497, -0.795912, 1.570796, 1.688669],accel_mss,speed_ms,0,blend_radius_m)
    movel([0.117791, -1.283772, -2.632616, -0.796000, 1.570796, 1.688587],accel_mss,speed_ms,0,blend_radius_m)
    movel([0.117513, -1.284070, -2.632445, -0.795874, 1.570796, 1.688309],accel_mss,speed_ms,0,blend_radius_m)
    movel([0.117263, -1.284026, -2.632470, -0.795893, 1.570796, 1.688060],accel_mss,speed_ms,0,blend_radius_m)
    movel([0.116775, -1.283947, -2.632515, -0.795926, 1.570796, 1.687571],accel_mss,speed_ms,0,blend_radius_m)
    movel([0.116521, -1.283710, -2.632652, -0.796027, 1.570796, 1.687318],accel_mss,speed_ms,0,blend_radius_m)
    movel([0.116399, -1.283433, -2.632811, -0.796145, 1.570796, 1.687195],accel_mss,speed_ms,0,blend_radius_m)
    movel([0.116380, -1.283147, -2.632976, -0.796266, 1.570796, 1.687176],accel_mss,speed_ms,0,blend_radius_m)
    movel([0.116535, -1.282859, -2.633141, -0.796389, 1.570796, 1.687332],accel_mss,speed_ms,0,blend_radius_m)
    movel([0.116603, -1.283081, -2.633014, -0.796295, 1.570796, 1.687400],accel_mss,speed_ms,0,blend_radius_m)
    movel([0.116900, -1.282844, -2.633150, -0.796395, 1.570796, 1.687696],accel_mss,speed_ms,0,blend_radius_m)
    movel([0.116924, -1.282576, -2.633304, -0.796510, 1.570796, 1.687721],accel_mss,speed_ms,0,blend_radius_m)
    movel([0.116662, -1.282485, -2.633355, -0.796548, 1.570796, 1.687458],accel_mss,speed_ms,0,blend_radius_m)
    movel([0.117083, -1.282291, -2.633467, -0.796631, 1.570796, 1.687879],accel_mss,speed_ms,0,blend_radius_m)
    movel([0.117398, -1.282179, -2.633531, -0.796679, 1.570796, 1.688195],accel_mss,speed_ms,0,blend_radius_m)
    movel([0.117220, -1.281984, -2.633643, -0.796762, 1.570796, 1.688016],accel_mss,speed_ms,0,blend_radius_m)
    movel([0.116901, -1.282160, -2.633542, -0.796687, 1.570796, 1.687697],accel_mss,speed_ms,0,blend_radius_m)
    movel([0.117066, -1.281823, -2.633735, -0.796831, 1.570796, 1.687862],accel_mss,speed_ms,0,blend_radius_m)
    movel([0.117091, -1.281486, -2.633928, -0.796975, 1.570796, 1.687888],accel_mss,speed_ms,0,blend_radius_m)
    movel([0.117345, -1.281132, -2.634131, -0.797127, 1.570796, 1.688141],accel_mss,speed_ms,0,blend_radius_m)
    movel([0.117730, -1.281234, -2.634072, -0.797083, 1.570796, 1.688526],accel_mss,speed_ms,0,blend_radius_m)
    movel([0.117907, -1.281357, -2.634002, -0.797030, 1.570796, 1.688704],accel_mss,speed_ms,0,blend_radius_m)
    movel([0.118256, -1.281123, -2.634136, -0.797130, 1.570796, 1.689052],accel_mss,speed_ms,0,blend_radius_m)
    movel([0.118549, -1.281003, -2.634204, -0.797182, 1.570796, 1.689345],accel_mss,speed_ms,0,blend_radius_m)
    movel([0.118546, -1.280735, -2.634357, -0.797296, 1.570796, 1.689343],accel_mss,speed_ms,0,blend_radius_m)
    movel([0.118238, -1.280647, -2.634408, -0.797334, 1.570796, 1.689034],accel_mss,speed_ms,0,blend_radius_m)
    movel([0.117886, -1.280906, -2.634259, -0.797223, 1.570796, 1.688682],accel_mss,speed_ms,0,blend_radius_m)
    movel([0.117733, -1.280735, -2.634358, -0.797297, 1.570796, 1.688530],accel_mss,speed_ms,0,blend_radius_m)
    movel([0.117417, -1.280828, -2.634304, -0.797257, 1.570796, 1.688213],accel_mss,speed_ms,0,blend_radius_m)
    movel([0.117154, -1.280801, -2.634320, -0.797269, 1.570796, 1.687950],accel_mss,speed_ms,0,blend_radius_m)
    movel([0.117279, -1.280976, -2.634220, -0.797193, 1.570796, 1.688075],accel_mss,speed_ms,0,blend_radius_m)
    movel([0.117007, -1.281203, -2.634090, -0.797096, 1.570796, 1.687803],accel_mss,speed_ms,0,blend_radius_m)
    movel([0.116841, -1.280946, -2.634237, -0.797206, 1.570796, 1.687638],accel_mss,speed_ms,0,blend_radius_m)
    movel([0.116572, -1.280906, -2.634259, -0.797223, 1.570796, 1.687368],accel_mss,speed_ms,0,blend_radius_m)
    movel([0.116208, -1.280785, -2.634329, -0.797275, 1.570796, 1.687004],accel_mss,speed_ms,0,blend_radius_m)
    movel([0.116016, -1.280684, -2.634386, -0.797318, 1.570796, 1.686813],accel_mss,speed_ms,0,blend_radius_m)
    movel([0.115720, -1.280479, -2.634504, -0.797406, 1.570796, 1.686516],accel_mss,speed_ms,0,blend_radius_m)
    movel([0.115647, -1.280267, -2.634624, -0.797497, 1.570796, 1.686444],accel_mss,speed_ms,0,blend_radius_m)
    movel([0.115443, -1.280134, -2.634701, -0.797554, 1.570796, 1.686240],accel_mss,speed_ms,0,blend_radius_m)
    movel([0.115403, -1.280409, -2.634544, -0.797437, 1.570796, 1.686199],accel_mss,speed_ms,0,blend_radius_m)
    movel([0.115514, -1.280613, -2.634427, -0.797349, 1.570796, 1.686310],accel_mss,speed_ms,0,blend_radius_m)
    movel([0.115629, -1.280801, -2.634320, -0.797268, 1.570796, 1.686426],accel_mss,speed_ms,0,blend_radius_m)
    movel([0.115390, -1.281049, -2.634178, -0.797162, 1.570796, 1.686186],accel_mss,speed_ms,0,blend_radius_m)
    movel([0.115503, -1.280762, -2.634342, -0.797285, 1.570796, 1.686299],accel_mss,speed_ms,0,blend_radius_m)
    movel([0.115218, -1.280712, -2.634370, -0.797306, 1.570796, 1.686014],accel_mss,speed_ms,0,blend_radius_m)
    movel([0.115021, -1.280548, -2.634464, -0.797377, 1.570796, 1.685817],accel_mss,speed_ms,0,blend_radius_m)
    movel([0.115096, -1.280190, -2.634669, -0.797531, 1.570796, 1.685893],accel_mss,speed_ms,0,blend_radius_m)
    movel([0.115346, -1.279945, -2.634809, -0.797636, 1.570796, 1.686143],accel_mss,speed_ms,0,blend_radius_m)
    movel([0.115659, -1.279760, -2.634914, -0.797715, 1.570796, 1.686455],accel_mss,speed_ms,0,blend_radius_m)
    movel([0.115744, -1.279475, -2.635076, -0.797838, 1.570796, 1.686541],accel_mss,speed_ms,0,blend_radius_m)
    movel([0.115466, -1.279480, -2.635074, -0.797836, 1.570796, 1.686262],accel_mss,speed_ms,0,blend_radius_m)
    movel([0.115654, -1.279611, -2.634999, -0.797779, 1.570796, 1.686450],accel_mss,speed_ms,0,blend_radius_m)
    movel([0.115361, -1.279773, -2.634907, -0.797710, 1.570796, 1.686157],accel_mss,speed_ms,0,blend_radius_m)
    movel([0.115061, -1.280005, -2.634774, -0.797610, 1.570796, 1.685857],accel_mss,speed_ms,0,blend_radius_m)
    movel([0.115080, -1.279688, -2.634955, -0.797746, 1.570796, 1.685876],accel_mss,speed_ms,0,blend_radius_m)
    movel([0.115258, -1.279309, -2.635171, -0.797909, 1.570796, 1.686055],accel_mss,speed_ms,0,blend_radius_m)
    movel([0.115654, -1.278752, -2.635488, -0.798149, 1.570796, 1.686451],accel_mss,speed_ms,0,blend_radius_m)
    movel([0.116074, -1.278243, -2.635777, -0.798369, 1.570796, 1.686870],accel_mss,speed_ms,0,blend_radius_m)
    movel([0.116426, -1.278050, -2.635887, -0.798452, 1.570796, 1.687222],accel_mss,speed_ms,0,blend_radius_m)
    movel([0.116646, -1.277773, -2.636044, -0.798572, 1.570796, 1.687442],accel_mss,speed_ms,0,blend_radius_m)
    movel([0.116582, -1.278078, -2.635871, -0.798440, 1.570796, 1.687378],accel_mss,speed_ms,0,blend_radius_m)
    movel([0.116643, -1.278294, -2.635748, -0.798347, 1.570796, 1.687439],accel_mss,speed_ms,0,blend_radius_m)
    movel([0.116707, -1.278011, -2.635909, -0.798469, 1.570796, 1.687503],accel_mss,speed_ms,0,blend_radius_m)
    movel([0.116909, -1.277684, -2.636095, -0.798610, 1.570796, 1.687705],accel_mss,speed_ms,0,blend_radius_m)
    movel([0.117205, -1.277277, -2.636325, -0.798786, 1.570796, 1.688001],accel_mss,speed_ms,0,blend_radius_m)
    movel([0.117543, -1.276945, -2.636514, -0.798930, 1.570796, 1.688340],accel_mss,speed_ms,0,blend_radius_m)
    movel([0.117995, -1.276571, -2.636726, -0.799092, 1.570796, 1.688792],accel_mss,speed_ms,0,blend_radius_m)
    movel([0.118505, -1.276213, -2.636928, -0.799248, 1.570796, 1.689301],accel_mss,speed_ms,0,blend_radius_m)
    movel([0.118905, -1.276012, -2.637042, -0.799335, 1.570796, 1.689701],accel_mss,speed_ms,0,blend_radius_m)
    movel([0.119186, -1.275854, -2.637131, -0.799404, 1.570796, 1.689982],accel_mss,speed_ms,0,blend_radius_m)
    movel([0.119588, -1.275394, -2.637391, -0.799604, 1.570796, 1.690384],accel_mss,speed_ms,0,blend_radius_m)
    movel([0.120097, -1.275070, -2.637574, -0.799745, 1.570796, 1.690893],accel_mss,speed_ms,0,blend_radius_m)
    movel([0.120709, -1.274745, -2.637757, -0.799887, 1.570796, 1.691505],accel_mss,speed_ms,0,blend_radius_m)
    speed_ms = 0.003
    movel([0.120709, -1.278294, -2.639421, -0.794674, 1.570796, 1.691505],accel_mss,speed_ms,0,blend_radius_m)
    speed_ms = 0.007
    movel([0.121089, -1.278104, -2.639528, -0.794756, 1.570796, 1.691885],accel_mss,speed_ms,0,blend_radius_m)
